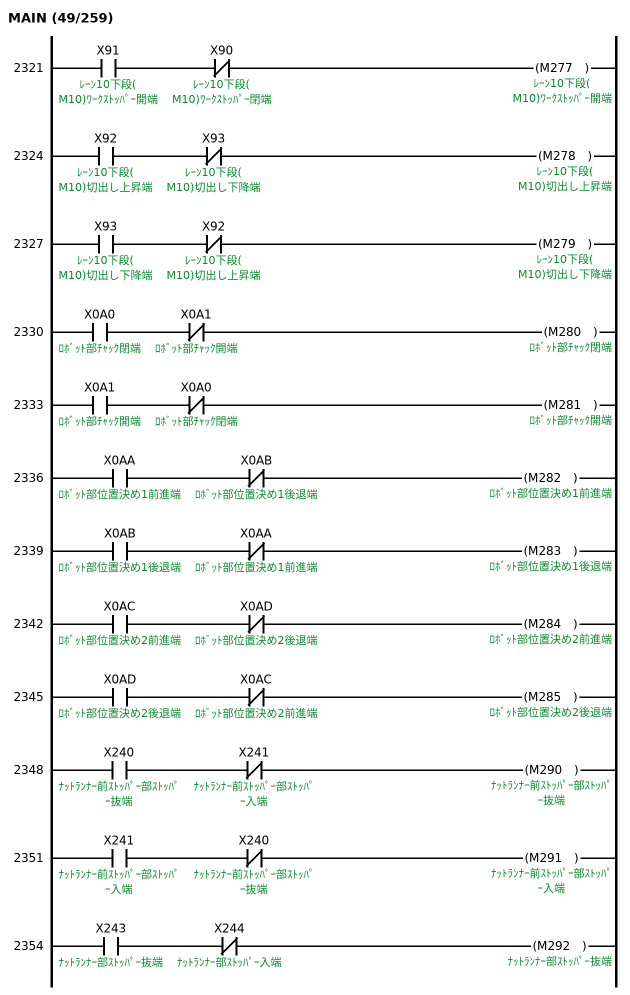
[picture p48: ladder of MAIN, rungs at steps 2321 to 2354]
2321  LD      X91  ; ﾚｰﾝ10下段(M10)ﾜｰｸｽﾄｯﾊﾟｰ開端
      ANI     X90  ; ﾚｰﾝ10下段(M10)ﾜｰｸｽﾄｯﾊﾟｰ閉端
      OUT     M277  ; ﾚｰﾝ10下段(M10)ﾜｰｸｽﾄｯﾊﾟｰ開端
2324  LD      X92  ; ﾚｰﾝ10下段(M10)切出し上昇端
      ANI     X93  ; ﾚｰﾝ10下段(M10)切出し下降端
      OUT     M278  ; ﾚｰﾝ10下段(M10)切出し上昇端
2327  LD      X93  ; ﾚｰﾝ10下段(M10)切出し下降端
      ANI     X92  ; ﾚｰﾝ10下段(M10)切出し上昇端
      OUT     M279  ; ﾚｰﾝ10下段(M10)切出し下降端
2330  LD      X0A0  ; ﾛﾎﾞｯﾄ部ﾁｬｯｸ閉端
      ANI     X0A1  ; ﾛﾎﾞｯﾄ部ﾁｬｯｸ開端
      OUT     M280  ; ﾛﾎﾞｯﾄ部ﾁｬｯｸ閉端
2333  LD      X0A1  ; ﾛﾎﾞｯﾄ部ﾁｬｯｸ開端
      ANI     X0A0  ; ﾛﾎﾞｯﾄ部ﾁｬｯｸ閉端
      OUT     M281  ; ﾛﾎﾞｯﾄ部ﾁｬｯｸ開端
2336  LD      X0AA  ; ﾛﾎﾞｯﾄ部位置決め1前進端
      ANI     X0AB  ; ﾛﾎﾞｯﾄ部位置決め1後退端
      OUT     M282  ; ﾛﾎﾞｯﾄ部位置決め1前進端
2339  LD      X0AB  ; ﾛﾎﾞｯﾄ部位置決め1後退端
      ANI     X0AA  ; ﾛﾎﾞｯﾄ部位置決め1前進端
      OUT     M283  ; ﾛﾎﾞｯﾄ部位置決め1後退端
2342  LD      X0AC  ; ﾛﾎﾞｯﾄ部位置決め2前進端
      ANI     X0AD  ; ﾛﾎﾞｯﾄ部位置決め2後退端
      OUT     M284  ; ﾛﾎﾞｯﾄ部位置決め2前進端
2345  LD      X0AD  ; ﾛﾎﾞｯﾄ部位置決め2後退端
      ANI     X0AC  ; ﾛﾎﾞｯﾄ部位置決め2前進端
      OUT     M285  ; ﾛﾎﾞｯﾄ部位置決め2後退端
2348  LD      X240  ; ﾅｯﾄﾗﾝﾅｰ前ｽﾄｯﾊﾟｰ部ｽﾄｯﾊﾟｰ抜端
      ANI     X241  ; ﾅｯﾄﾗﾝﾅｰ前ｽﾄｯﾊﾟｰ部ｽﾄｯﾊﾟｰ入端
      OUT     M290  ; ﾅｯﾄﾗﾝﾅｰ前ｽﾄｯﾊﾟｰ部ｽﾄｯﾊﾟｰ抜端
2351  LD      X241  ; ﾅｯﾄﾗﾝﾅｰ前ｽﾄｯﾊﾟｰ部ｽﾄｯﾊﾟｰ入端
      ANI     X240  ; ﾅｯﾄﾗﾝﾅｰ前ｽﾄｯﾊﾟｰ部ｽﾄｯﾊﾟｰ抜端
      OUT     M291  ; ﾅｯﾄﾗﾝﾅｰ前ｽﾄｯﾊﾟｰ部ｽﾄｯﾊﾟｰ入端
2354  LD      X243  ; ﾅｯﾄﾗﾝﾅｰ部ｽﾄｯﾊﾟｰ抜端
      ANI     X244  ; ﾅｯﾄﾗﾝﾅｰ部ｽﾄｯﾊﾟｰ入端
      OUT     M292  ; ﾅｯﾄﾗﾝﾅｰ部ｽﾄｯﾊﾟｰ抜端
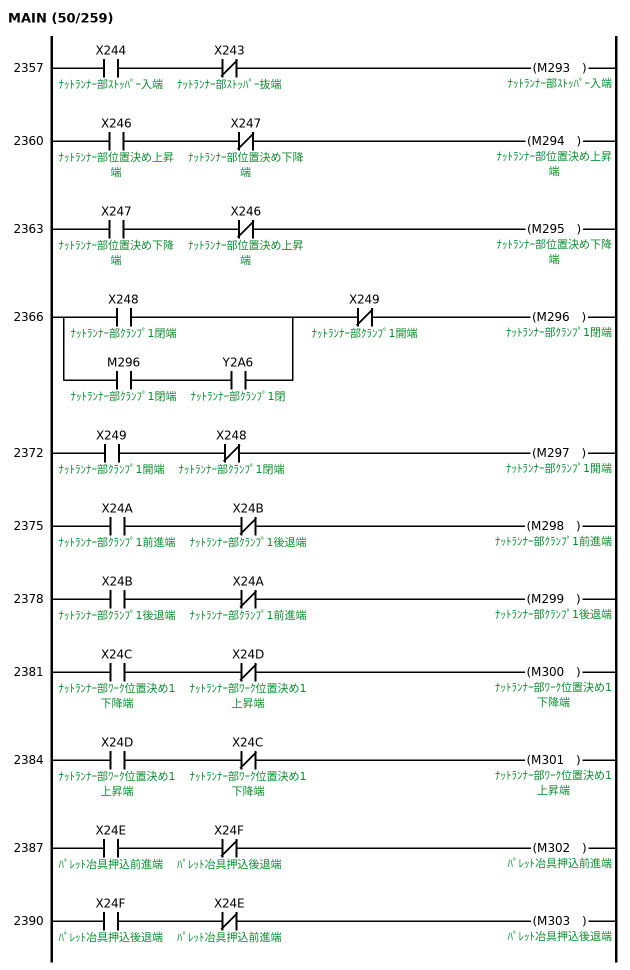
2357  LD      X244  ; ﾅｯﾄﾗﾝﾅｰ部ｽﾄｯﾊﾟｰ入端
      ANI     X243  ; ﾅｯﾄﾗﾝﾅｰ部ｽﾄｯﾊﾟｰ抜端
      OUT     M293  ; ﾅｯﾄﾗﾝﾅｰ部ｽﾄｯﾊﾟｰ入端
2360  LD      X246  ; ﾅｯﾄﾗﾝﾅｰ部位置決め上昇端
      ANI     X247  ; ﾅｯﾄﾗﾝﾅｰ部位置決め下降端
      OUT     M294  ; ﾅｯﾄﾗﾝﾅｰ部位置決め上昇端
2363  LD      X247  ; ﾅｯﾄﾗﾝﾅｰ部位置決め下降端
      ANI     X246  ; ﾅｯﾄﾗﾝﾅｰ部位置決め上昇端
      OUT     M295  ; ﾅｯﾄﾗﾝﾅｰ部位置決め下降端
2366  LD      X248  ; ﾅｯﾄﾗﾝﾅｰ部ｸﾗﾝﾌﾟ1閉端
      LD      M296  ; ﾅｯﾄﾗﾝﾅｰ部ｸﾗﾝﾌﾟ1閉端
      AND     Y2A6  ; ﾅｯﾄﾗﾝﾅｰ部ｸﾗﾝﾌﾟ1閉
      ORB
      ANI     X249  ; ﾅｯﾄﾗﾝﾅｰ部ｸﾗﾝﾌﾟ1開端
      OUT     M296  ; ﾅｯﾄﾗﾝﾅｰ部ｸﾗﾝﾌﾟ1閉端
2372  LD      X249  ; ﾅｯﾄﾗﾝﾅｰ部ｸﾗﾝﾌﾟ1開端
      ANI     X248  ; ﾅｯﾄﾗﾝﾅｰ部ｸﾗﾝﾌﾟ1閉端
      OUT     M297  ; ﾅｯﾄﾗﾝﾅｰ部ｸﾗﾝﾌﾟ1開端
2375  LD      X24A  ; ﾅｯﾄﾗﾝﾅｰ部ｸﾗﾝﾌﾟ1前進端
      ANI     X24B  ; ﾅｯﾄﾗﾝﾅｰ部ｸﾗﾝﾌﾟ1後退端
      OUT     M298  ; ﾅｯﾄﾗﾝﾅｰ部ｸﾗﾝﾌﾟ1前進端
2378  LD      X24B  ; ﾅｯﾄﾗﾝﾅｰ部ｸﾗﾝﾌﾟ1後退端
      ANI     X24A  ; ﾅｯﾄﾗﾝﾅｰ部ｸﾗﾝﾌﾟ1前進端
      OUT     M299  ; ﾅｯﾄﾗﾝﾅｰ部ｸﾗﾝﾌﾟ1後退端
2381  LD      X24C  ; ﾅｯﾄﾗﾝﾅｰ部ﾜｰｸ位置決め1下降端
      ANI     X24D  ; ﾅｯﾄﾗﾝﾅｰ部ﾜｰｸ位置決め1上昇端
      OUT     M300  ; ﾅｯﾄﾗﾝﾅｰ部ﾜｰｸ位置決め1下降端
2384  LD      X24D  ; ﾅｯﾄﾗﾝﾅｰ部ﾜｰｸ位置決め1上昇端
      ANI     X24C  ; ﾅｯﾄﾗﾝﾅｰ部ﾜｰｸ位置決め1下降端
      OUT     M301  ; ﾅｯﾄﾗﾝﾅｰ部ﾜｰｸ位置決め1上昇端
2387  LD      X24E  ; ﾊﾟﾚｯﾄ冶具押込前進端
      ANI     X24F  ; ﾊﾟﾚｯﾄ冶具押込後退端
      OUT     M302  ; ﾊﾟﾚｯﾄ冶具押込前進端
2390  LD      X24F  ; ﾊﾟﾚｯﾄ冶具押込後退端
      ANI     X24E  ; ﾊﾟﾚｯﾄ冶具押込前進端
      OUT     M303  ; ﾊﾟﾚｯﾄ冶具押込後退端
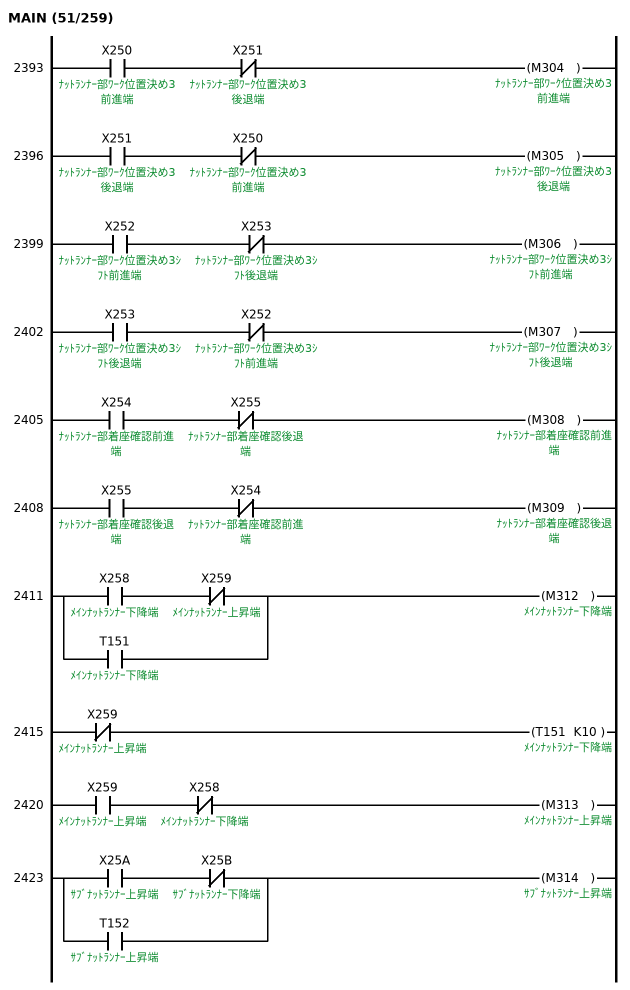
2393  LD      X250  ; ﾅｯﾄﾗﾝﾅｰ部ﾜｰｸ位置決め3前進端
      ANI     X251  ; ﾅｯﾄﾗﾝﾅｰ部ﾜｰｸ位置決め3後退端
      OUT     M304  ; ﾅｯﾄﾗﾝﾅｰ部ﾜｰｸ位置決め3前進端
2396  LD      X251  ; ﾅｯﾄﾗﾝﾅｰ部ﾜｰｸ位置決め3後退端
      ANI     X250  ; ﾅｯﾄﾗﾝﾅｰ部ﾜｰｸ位置決め3前進端
      OUT     M305  ; ﾅｯﾄﾗﾝﾅｰ部ﾜｰｸ位置決め3後退端
2399  LD      X252  ; ﾅｯﾄﾗﾝﾅｰ部ﾜｰｸ位置決め3ｼﾌﾄ前進端
      ANI     X253  ; ﾅｯﾄﾗﾝﾅｰ部ﾜｰｸ位置決め3ｼﾌﾄ後退端
      OUT     M306  ; ﾅｯﾄﾗﾝﾅｰ部ﾜｰｸ位置決め3ｼﾌﾄ前進端
2402  LD      X253  ; ﾅｯﾄﾗﾝﾅｰ部ﾜｰｸ位置決め3ｼﾌﾄ後退端
      ANI     X252  ; ﾅｯﾄﾗﾝﾅｰ部ﾜｰｸ位置決め3ｼﾌﾄ前進端
      OUT     M307  ; ﾅｯﾄﾗﾝﾅｰ部ﾜｰｸ位置決め3ｼﾌﾄ後退端
2405  LD      X254  ; ﾅｯﾄﾗﾝﾅｰ部着座確認前進端
      ANI     X255  ; ﾅｯﾄﾗﾝﾅｰ部着座確認後退端
      OUT     M308  ; ﾅｯﾄﾗﾝﾅｰ部着座確認前進端
2408  LD      X255  ; ﾅｯﾄﾗﾝﾅｰ部着座確認後退端
      ANI     X254  ; ﾅｯﾄﾗﾝﾅｰ部着座確認前進端
      OUT     M309  ; ﾅｯﾄﾗﾝﾅｰ部着座確認後退端
2411  LD      X258  ; ﾒｲﾝﾅｯﾄﾗﾝﾅｰ下降端
      ANI     X259  ; ﾒｲﾝﾅｯﾄﾗﾝﾅｰ上昇端
      OR      T151  ; ﾒｲﾝﾅｯﾄﾗﾝﾅｰ下降端
      OUT     M312  ; ﾒｲﾝﾅｯﾄﾗﾝﾅｰ下降端
2415  LDI     X259  ; ﾒｲﾝﾅｯﾄﾗﾝﾅｰ上昇端
      OUT     T151 K10  ; ﾒｲﾝﾅｯﾄﾗﾝﾅｰ下降端
2420  LD      X259  ; ﾒｲﾝﾅｯﾄﾗﾝﾅｰ上昇端
      ANI     X258  ; ﾒｲﾝﾅｯﾄﾗﾝﾅｰ下降端
      OUT     M313  ; ﾒｲﾝﾅｯﾄﾗﾝﾅｰ上昇端
2423  LD      X25A  ; ｻﾌﾞﾅｯﾄﾗﾝﾅｰ上昇端
      ANI     X25B  ; ｻﾌﾞﾅｯﾄﾗﾝﾅｰ下降端
      OR      T152  ; ｻﾌﾞﾅｯﾄﾗﾝﾅｰ上昇端
      OUT     M314  ; ｻﾌﾞﾅｯﾄﾗﾝﾅｰ上昇端
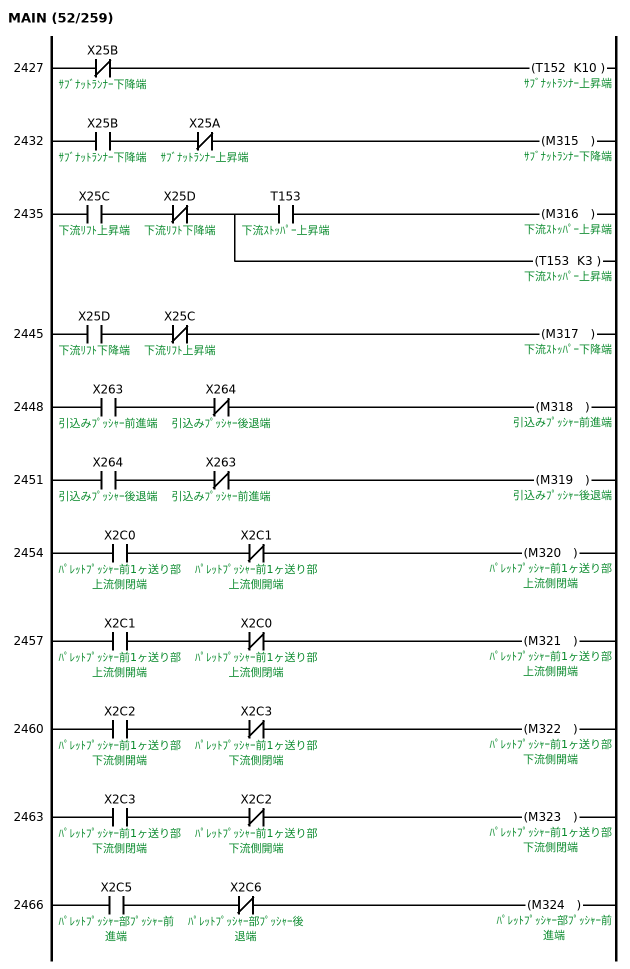
2427  LDI     X25B  ; ｻﾌﾞﾅｯﾄﾗﾝﾅｰ下降端
      OUT     T152 K10  ; ｻﾌﾞﾅｯﾄﾗﾝﾅｰ上昇端
2432  LD      X25B  ; ｻﾌﾞﾅｯﾄﾗﾝﾅｰ下降端
      ANI     X25A  ; ｻﾌﾞﾅｯﾄﾗﾝﾅｰ上昇端
      OUT     M315  ; ｻﾌﾞﾅｯﾄﾗﾝﾅｰ下降端
2435  LD      X25C  ; 下流ﾘﾌﾄ上昇端
      ANI     X25D  ; 下流ﾘﾌﾄ下降端
      MPS
      AND     T153  ; 下流ｽﾄｯﾊﾟｰ上昇端
      OUT     M316  ; 下流ｽﾄｯﾊﾟｰ上昇端
      MPP
      OUT     T153 K3  ; 下流ｽﾄｯﾊﾟｰ上昇端
2445  LD      X25D  ; 下流ﾘﾌﾄ下降端
      ANI     X25C  ; 下流ﾘﾌﾄ上昇端
      OUT     M317  ; 下流ｽﾄｯﾊﾟｰ下降端
2448  LD      X263  ; 引込みﾌﾟｯｼｬｰ前進端
      ANI     X264  ; 引込みﾌﾟｯｼｬｰ後退端
      OUT     M318  ; 引込みﾌﾟｯｼｬｰ前進端
2451  LD      X264  ; 引込みﾌﾟｯｼｬｰ後退端
      ANI     X263  ; 引込みﾌﾟｯｼｬｰ前進端
      OUT     M319  ; 引込みﾌﾟｯｼｬｰ後退端
2454  LD      X2C0  ; ﾊﾟﾚｯﾄﾌﾟｯｼｬｰ前1ヶ送り部上流側閉端
      ANI     X2C1  ; ﾊﾟﾚｯﾄﾌﾟｯｼｬｰ前1ヶ送り部上流側開端
      OUT     M320  ; ﾊﾟﾚｯﾄﾌﾟｯｼｬｰ前1ヶ送り部上流側閉端
2457  LD      X2C1  ; ﾊﾟﾚｯﾄﾌﾟｯｼｬｰ前1ヶ送り部上流側開端
      ANI     X2C0  ; ﾊﾟﾚｯﾄﾌﾟｯｼｬｰ前1ヶ送り部上流側閉端
      OUT     M321  ; ﾊﾟﾚｯﾄﾌﾟｯｼｬｰ前1ヶ送り部上流側開端
2460  LD      X2C2  ; ﾊﾟﾚｯﾄﾌﾟｯｼｬｰ前1ヶ送り部下流側開端
      ANI     X2C3  ; ﾊﾟﾚｯﾄﾌﾟｯｼｬｰ前1ヶ送り部下流側閉端
      OUT     M322  ; ﾊﾟﾚｯﾄﾌﾟｯｼｬｰ前1ヶ送り部下流側開端
2463  LD      X2C3  ; ﾊﾟﾚｯﾄﾌﾟｯｼｬｰ前1ヶ送り部下流側閉端
      ANI     X2C2  ; ﾊﾟﾚｯﾄﾌﾟｯｼｬｰ前1ヶ送り部下流側開端
      OUT     M323  ; ﾊﾟﾚｯﾄﾌﾟｯｼｬｰ前1ヶ送り部下流側閉端
2466  LD      X2C5  ; ﾊﾟﾚｯﾄﾌﾟｯｼｬｰ部ﾌﾟｯｼｬｰ前進端
      ANI     X2C6  ; ﾊﾟﾚｯﾄﾌﾟｯｼｬｰ部ﾌﾟｯｼｬｰ後退端
      OUT     M324  ; ﾊﾟﾚｯﾄﾌﾟｯｼｬｰ部ﾌﾟｯｼｬｰ前進端
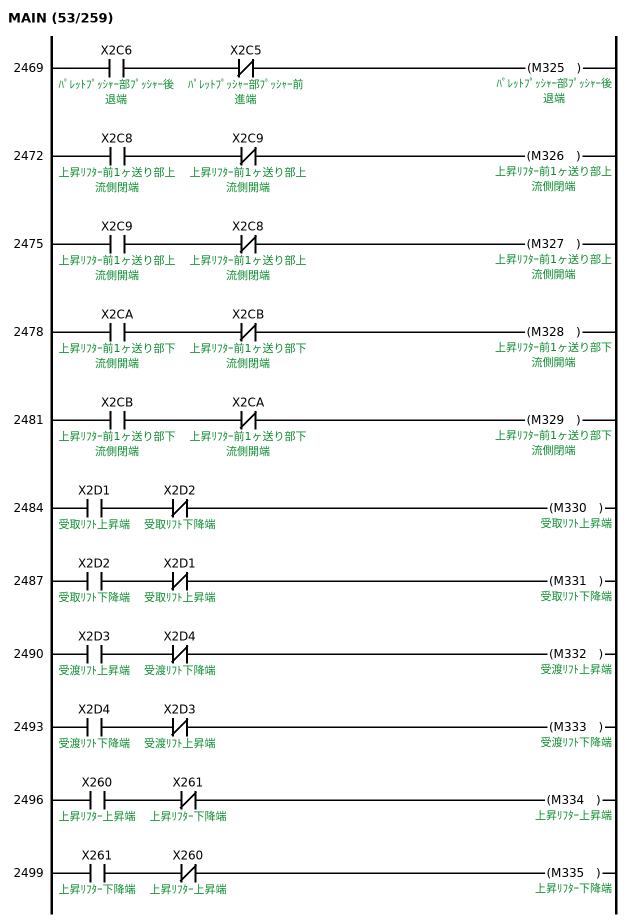
2469  LD      X2C6  ; ﾊﾟﾚｯﾄﾌﾟｯｼｬｰ部ﾌﾟｯｼｬｰ後退端
      ANI     X2C5  ; ﾊﾟﾚｯﾄﾌﾟｯｼｬｰ部ﾌﾟｯｼｬｰ前進端
      OUT     M325  ; ﾊﾟﾚｯﾄﾌﾟｯｼｬｰ部ﾌﾟｯｼｬｰ後退端
2472  LD      X2C8  ; 上昇ﾘﾌﾀｰ前1ヶ送り部上流側閉端
      ANI     X2C9  ; 上昇ﾘﾌﾀｰ前1ヶ送り部上流側開端
      OUT     M326  ; 上昇ﾘﾌﾀｰ前1ヶ送り部上流側閉端
2475  LD      X2C9  ; 上昇ﾘﾌﾀｰ前1ヶ送り部上流側開端
      ANI     X2C8  ; 上昇ﾘﾌﾀｰ前1ヶ送り部上流側閉端
      OUT     M327  ; 上昇ﾘﾌﾀｰ前1ヶ送り部上流側開端
2478  LD      X2CA  ; 上昇ﾘﾌﾀｰ前1ヶ送り部下流側開端
      ANI     X2CB  ; 上昇ﾘﾌﾀｰ前1ヶ送り部下流側閉端
      OUT     M328  ; 上昇ﾘﾌﾀｰ前1ヶ送り部下流側開端
2481  LD      X2CB  ; 上昇ﾘﾌﾀｰ前1ヶ送り部下流側閉端
      ANI     X2CA  ; 上昇ﾘﾌﾀｰ前1ヶ送り部下流側開端
      OUT     M329  ; 上昇ﾘﾌﾀｰ前1ヶ送り部下流側閉端
2484  LD      X2D1  ; 受取ﾘﾌﾄ上昇端
      ANI     X2D2  ; 受取ﾘﾌﾄ下降端
      OUT     M330  ; 受取ﾘﾌﾄ上昇端
2487  LD      X2D2  ; 受取ﾘﾌﾄ下降端
      ANI     X2D1  ; 受取ﾘﾌﾄ上昇端
      OUT     M331  ; 受取ﾘﾌﾄ下降端
2490  LD      X2D3  ; 受渡ﾘﾌﾄ上昇端
      ANI     X2D4  ; 受渡ﾘﾌﾄ下降端
      OUT     M332  ; 受渡ﾘﾌﾄ上昇端
2493  LD      X2D4  ; 受渡ﾘﾌﾄ下降端
      ANI     X2D3  ; 受渡ﾘﾌﾄ上昇端
      OUT     M333  ; 受渡ﾘﾌﾄ下降端
2496  LD      X260  ; 上昇ﾘﾌﾀｰ上昇端
      ANI     X261  ; 上昇ﾘﾌﾀｰ下降端
      OUT     M334  ; 上昇ﾘﾌﾀｰ上昇端
2499  LD      X261  ; 上昇ﾘﾌﾀｰ下降端
      ANI     X260  ; 上昇ﾘﾌﾀｰ上昇端
      OUT     M335  ; 上昇ﾘﾌﾀｰ下降端
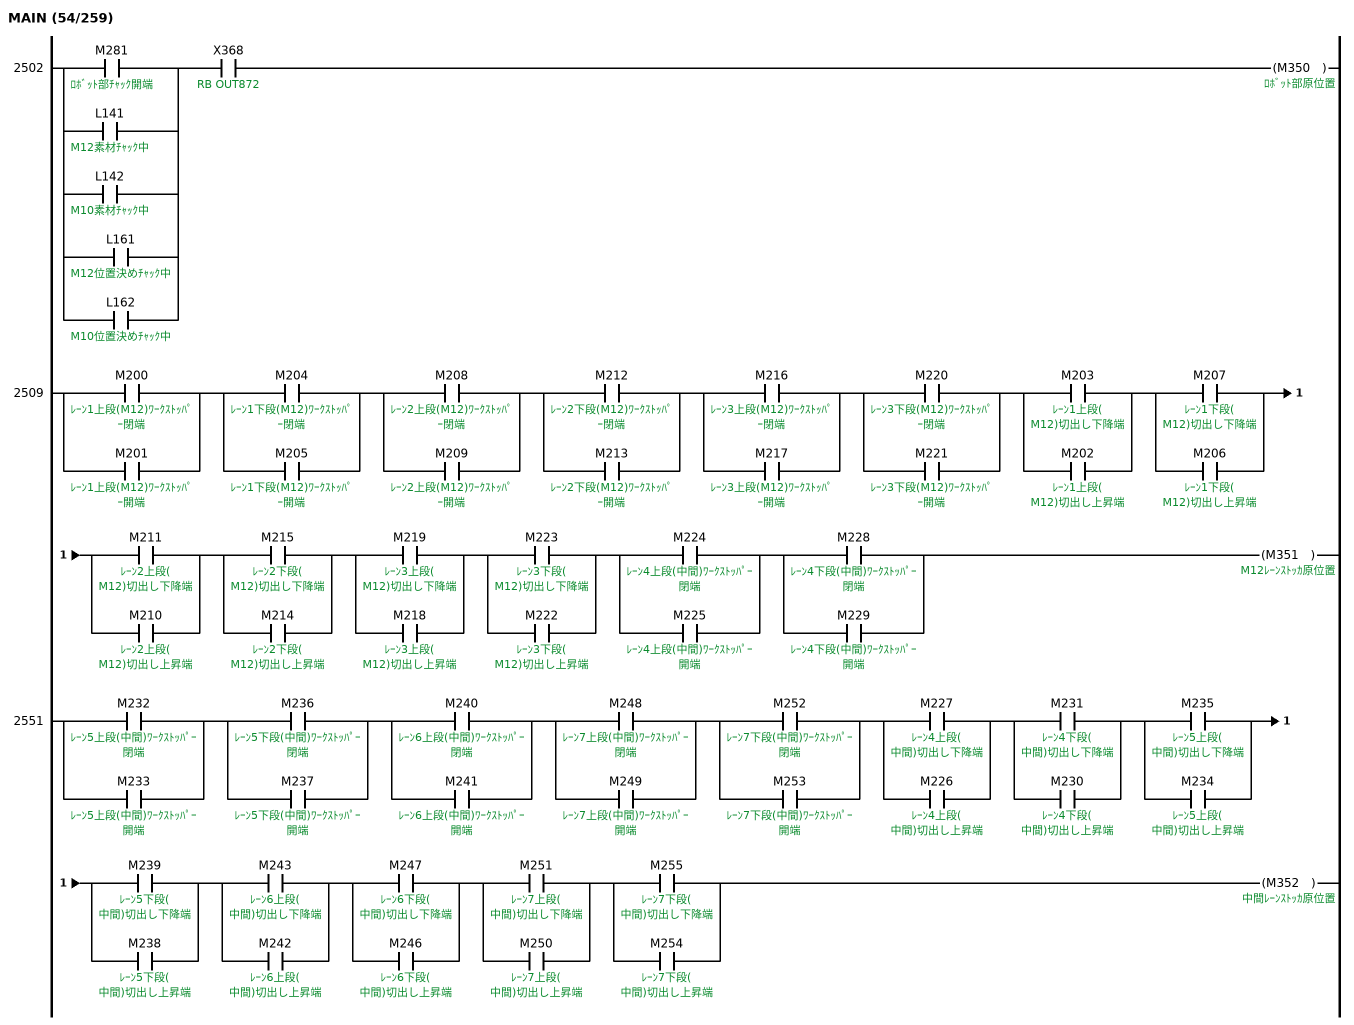
2502  LD      M281  ; ﾛﾎﾞｯﾄ部ﾁｬｯｸ開端
      OR      L141  ; M12素材ﾁｬｯｸ中
      OR      L142  ; M10素材ﾁｬｯｸ中
      OR      L161  ; M12位置決めﾁｬｯｸ中
      OR      L162  ; M10位置決めﾁｬｯｸ中
      AND     X368  ; RB OUT872
      OUT     M350  ; ﾛﾎﾞｯﾄ部原位置
2509  LD      M200  ; ﾚｰﾝ1上段(M12)ﾜｰｸｽﾄｯﾊﾟｰ閉端
      OR      M201  ; ﾚｰﾝ1上段(M12)ﾜｰｸｽﾄｯﾊﾟｰ開端
      LD      M204  ; ﾚｰﾝ1下段(M12)ﾜｰｸｽﾄｯﾊﾟｰ閉端
      OR      M205  ; ﾚｰﾝ1下段(M12)ﾜｰｸｽﾄｯﾊﾟｰ開端
      ANB
      LD      M208  ; ﾚｰﾝ2上段(M12)ﾜｰｸｽﾄｯﾊﾟｰ閉端
      OR      M209  ; ﾚｰﾝ2上段(M12)ﾜｰｸｽﾄｯﾊﾟｰ開端
      ANB
      LD      M212  ; ﾚｰﾝ2下段(M12)ﾜｰｸｽﾄｯﾊﾟｰ閉端
      OR      M213  ; ﾚｰﾝ2下段(M12)ﾜｰｸｽﾄｯﾊﾟｰ開端
      ANB
      LD      M216  ; ﾚｰﾝ3上段(M12)ﾜｰｸｽﾄｯﾊﾟｰ閉端
      OR      M217  ; ﾚｰﾝ3上段(M12)ﾜｰｸｽﾄｯﾊﾟｰ開端
      ANB
      LD      M220  ; ﾚｰﾝ3下段(M12)ﾜｰｸｽﾄｯﾊﾟｰ閉端
      OR      M221  ; ﾚｰﾝ3下段(M12)ﾜｰｸｽﾄｯﾊﾟｰ開端
      ANB
      LD      M203  ; ﾚｰﾝ1上段(M12)切出し下降端
      OR      M202  ; ﾚｰﾝ1上段(M12)切出し上昇端
      ANB
      LD      M207  ; ﾚｰﾝ1下段(M12)切出し下降端
      OR      M206  ; ﾚｰﾝ1下段(M12)切出し上昇端
      ANB
      LD      M211  ; ﾚｰﾝ2上段(M12)切出し下降端
      OR      M210  ; ﾚｰﾝ2上段(M12)切出し上昇端
      ANB
      LD      M215  ; ﾚｰﾝ2下段(M12)切出し下降端
      OR      M214  ; ﾚｰﾝ2下段(M12)切出し上昇端
      ANB
      LD      M219  ; ﾚｰﾝ3上段(M12)切出し下降端
      OR      M218  ; ﾚｰﾝ3上段(M12)切出し上昇端
      ANB
      LD      M223  ; ﾚｰﾝ3下段(M12)切出し下降端
      OR      M222  ; ﾚｰﾝ3下段(M12)切出し上昇端
      ANB
      LD      M224  ; ﾚｰﾝ4上段(中間)ﾜｰｸｽﾄｯﾊﾟｰ閉端
      OR      M225  ; ﾚｰﾝ4上段(中間)ﾜｰｸｽﾄｯﾊﾟｰ開端
      ANB
      LD      M228  ; ﾚｰﾝ4下段(中間)ﾜｰｸｽﾄｯﾊﾟｰ閉端
      OR      M229  ; ﾚｰﾝ4下段(中間)ﾜｰｸｽﾄｯﾊﾟｰ開端
      ANB
      OUT     M351  ; M12ﾚｰﾝｽﾄｯｶ原位置
2551  LD      M232  ; ﾚｰﾝ5上段(中間)ﾜｰｸｽﾄｯﾊﾟｰ閉端
      OR      M233  ; ﾚｰﾝ5上段(中間)ﾜｰｸｽﾄｯﾊﾟｰ開端
      LD      M236  ; ﾚｰﾝ5下段(中間)ﾜｰｸｽﾄｯﾊﾟｰ閉端
      OR      M237  ; ﾚｰﾝ5下段(中間)ﾜｰｸｽﾄｯﾊﾟｰ開端
      ANB
      LD      M240  ; ﾚｰﾝ6上段(中間)ﾜｰｸｽﾄｯﾊﾟｰ閉端
      OR      M241  ; ﾚｰﾝ6上段(中間)ﾜｰｸｽﾄｯﾊﾟｰ開端
      ANB
      LD      M248  ; ﾚｰﾝ7上段(中間)ﾜｰｸｽﾄｯﾊﾟｰ閉端
      OR      M249  ; ﾚｰﾝ7上段(中間)ﾜｰｸｽﾄｯﾊﾟｰ開端
      ANB
      LD      M252  ; ﾚｰﾝ7下段(中間)ﾜｰｸｽﾄｯﾊﾟｰ閉端
      OR      M253  ; ﾚｰﾝ7下段(中間)ﾜｰｸｽﾄｯﾊﾟｰ開端
      ANB
      LD      M227  ; ﾚｰﾝ4上段(中間)切出し下降端
      OR      M226  ; ﾚｰﾝ4上段(中間)切出し上昇端
      ANB
      LD      M231  ; ﾚｰﾝ4下段(中間)切出し下降端
      OR      M230  ; ﾚｰﾝ4下段(中間)切出し上昇端
      ANB
      LD      M235  ; ﾚｰﾝ5上段(中間)切出し下降端
      OR      M234  ; ﾚｰﾝ5上段(中間)切出し上昇端
      ANB
      LD      M239  ; ﾚｰﾝ5下段(中間)切出し下降端
      OR      M238  ; ﾚｰﾝ5下段(中間)切出し上昇端
      ANB
      LD      M243  ; ﾚｰﾝ6上段(中間)切出し下降端
      OR      M242  ; ﾚｰﾝ6上段(中間)切出し上昇端
      ANB
      LD      M247  ; ﾚｰﾝ6下段(中間)切出し下降端
      OR      M246  ; ﾚｰﾝ6下段(中間)切出し上昇端
      ANB
      LD      M251  ; ﾚｰﾝ7上段(中間)切出し下降端
      OR      M250  ; ﾚｰﾝ7上段(中間)切出し上昇端
      ANB
      LD      M255  ; ﾚｰﾝ7下段(中間)切出し下降端
      OR      M254  ; ﾚｰﾝ7下段(中間)切出し上昇端
      ANB
      OUT     M352  ; 中間ﾚｰﾝｽﾄｯｶ原位置
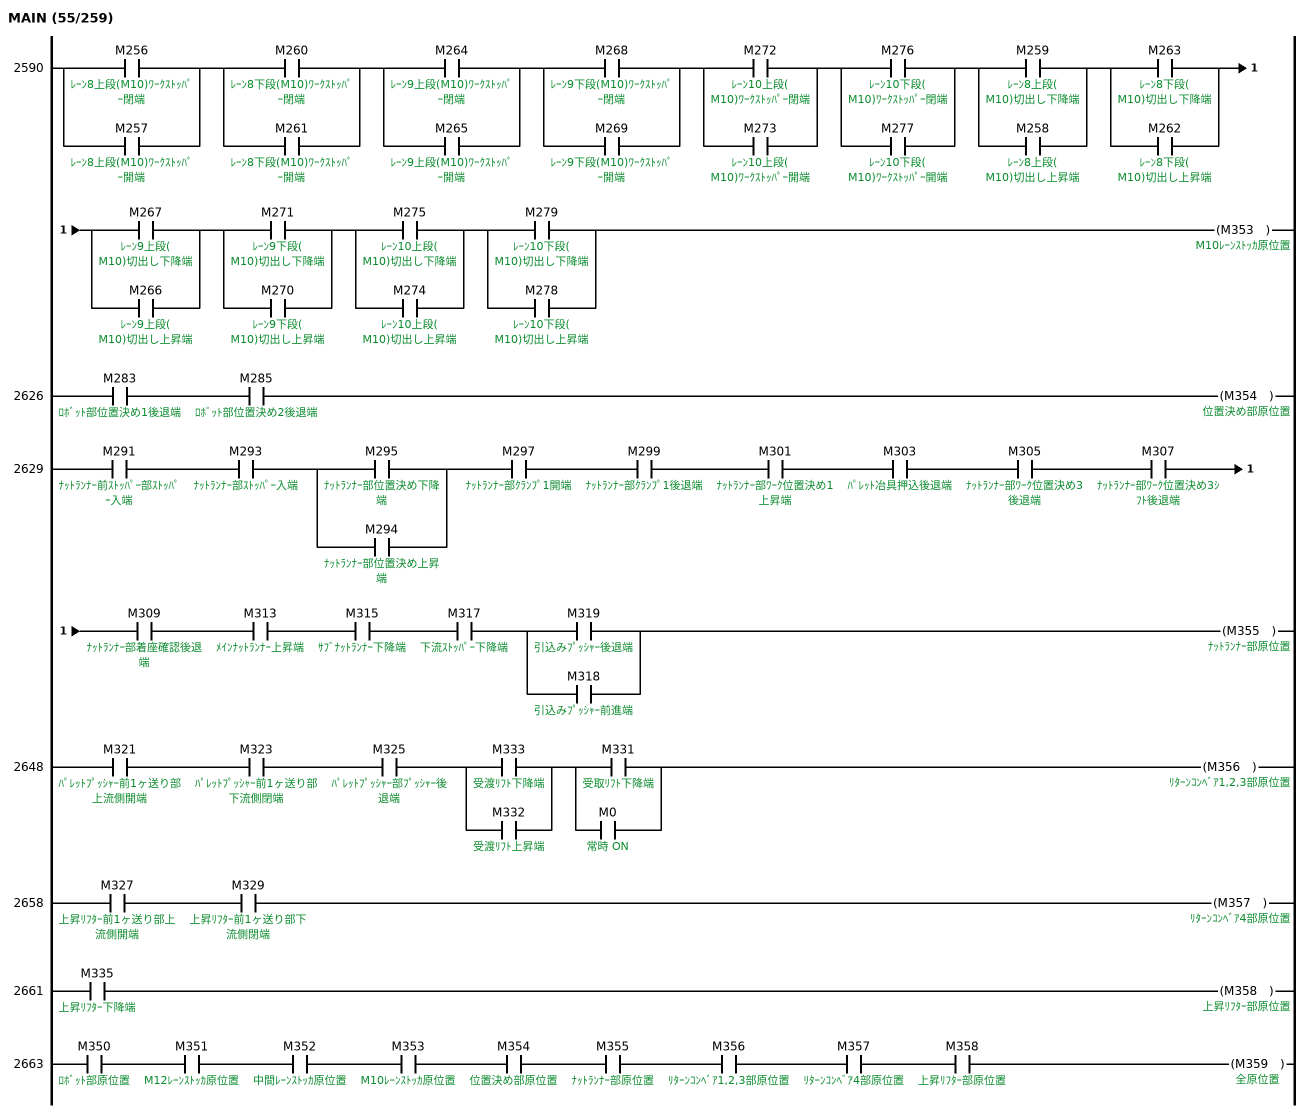
2590  LD      M256  ; ﾚｰﾝ8上段(M10)ﾜｰｸｽﾄｯﾊﾟｰ閉端
      OR      M257  ; ﾚｰﾝ8上段(M10)ﾜｰｸｽﾄｯﾊﾟｰ開端
      LD      M260  ; ﾚｰﾝ8下段(M10)ﾜｰｸｽﾄｯﾊﾟｰ閉端
      OR      M261  ; ﾚｰﾝ8下段(M10)ﾜｰｸｽﾄｯﾊﾟｰ開端
      ANB
      LD      M264  ; ﾚｰﾝ9上段(M10)ﾜｰｸｽﾄｯﾊﾟｰ閉端
      OR      M265  ; ﾚｰﾝ9上段(M10)ﾜｰｸｽﾄｯﾊﾟｰ開端
      ANB
      LD      M268  ; ﾚｰﾝ9下段(M10)ﾜｰｸｽﾄｯﾊﾟｰ閉端
      OR      M269  ; ﾚｰﾝ9下段(M10)ﾜｰｸｽﾄｯﾊﾟｰ開端
      ANB
      LD      M272  ; ﾚｰﾝ10上段(M10)ﾜｰｸｽﾄｯﾊﾟｰ閉端
      OR      M273  ; ﾚｰﾝ10上段(M10)ﾜｰｸｽﾄｯﾊﾟｰ開端
      ANB
      LD      M276  ; ﾚｰﾝ10下段(M10)ﾜｰｸｽﾄｯﾊﾟｰ閉端
      OR      M277  ; ﾚｰﾝ10下段(M10)ﾜｰｸｽﾄｯﾊﾟｰ開端
      ANB
      LD      M259  ; ﾚｰﾝ8上段(M10)切出し下降端
      OR      M258  ; ﾚｰﾝ8上段(M10)切出し上昇端
      ANB
      LD      M263  ; ﾚｰﾝ8下段(M10)切出し下降端
      OR      M262  ; ﾚｰﾝ8下段(M10)切出し上昇端
      ANB
      LD      M267  ; ﾚｰﾝ9上段(M10)切出し下降端
      OR      M266  ; ﾚｰﾝ9上段(M10)切出し上昇端
      ANB
      LD      M271  ; ﾚｰﾝ9下段(M10)切出し下降端
      OR      M270  ; ﾚｰﾝ9下段(M10)切出し上昇端
      ANB
      LD      M275  ; ﾚｰﾝ10上段(M10)切出し下降端
      OR      M274  ; ﾚｰﾝ10上段(M10)切出し上昇端
      ANB
      LD      M279  ; ﾚｰﾝ10下段(M10)切出し下降端
      OR      M278  ; ﾚｰﾝ10下段(M10)切出し上昇端
      ANB
      OUT     M353  ; M10ﾚｰﾝｽﾄｯｶ原位置
2626  LD      M283  ; ﾛﾎﾞｯﾄ部位置決め1後退端
      AND     M285  ; ﾛﾎﾞｯﾄ部位置決め2後退端
      OUT     M354  ; 位置決め部原位置
2629  LD      M291  ; ﾅｯﾄﾗﾝﾅｰ前ｽﾄｯﾊﾟｰ部ｽﾄｯﾊﾟｰ入端
      AND     M293  ; ﾅｯﾄﾗﾝﾅｰ部ｽﾄｯﾊﾟｰ入端
      LD      M295  ; ﾅｯﾄﾗﾝﾅｰ部位置決め下降端
      OR      M294  ; ﾅｯﾄﾗﾝﾅｰ部位置決め上昇端
      ANB
      AND     M297  ; ﾅｯﾄﾗﾝﾅｰ部ｸﾗﾝﾌﾟ1開端
      AND     M299  ; ﾅｯﾄﾗﾝﾅｰ部ｸﾗﾝﾌﾟ1後退端
      AND     M301  ; ﾅｯﾄﾗﾝﾅｰ部ﾜｰｸ位置決め1上昇端
      AND     M303  ; ﾊﾟﾚｯﾄ冶具押込後退端
      AND     M305  ; ﾅｯﾄﾗﾝﾅｰ部ﾜｰｸ位置決め3後退端
      AND     M307  ; ﾅｯﾄﾗﾝﾅｰ部ﾜｰｸ位置決め3ｼﾌﾄ後退端
      AND     M309  ; ﾅｯﾄﾗﾝﾅｰ部着座確認後退端
      AND     M313  ; ﾒｲﾝﾅｯﾄﾗﾝﾅｰ上昇端
      AND     M315  ; ｻﾌﾞﾅｯﾄﾗﾝﾅｰ下降端
      AND     M317  ; 下流ｽﾄｯﾊﾟｰ下降端
      LD      M319  ; 引込みﾌﾟｯｼｬｰ後退端
      OR      M318  ; 引込みﾌﾟｯｼｬｰ前進端
      ANB
      OUT     M355  ; ﾅｯﾄﾗﾝﾅｰ部原位置
2648  LD      M321  ; ﾊﾟﾚｯﾄﾌﾟｯｼｬｰ前1ヶ送り部上流側開端
      AND     M323  ; ﾊﾟﾚｯﾄﾌﾟｯｼｬｰ前1ヶ送り部下流側閉端
      AND     M325  ; ﾊﾟﾚｯﾄﾌﾟｯｼｬｰ部ﾌﾟｯｼｬｰ後退端
      LD      M333  ; 受渡ﾘﾌﾄ下降端
      OR      M332  ; 受渡ﾘﾌﾄ上昇端
      ANB
      LD      M331  ; 受取ﾘﾌﾄ下降端
      OR      M0  ; 常時 ON
      ANB
      OUT     M356  ; ﾘﾀｰﾝｺﾝﾍﾞｱ1,2,3部原位置
2658  LD      M327  ; 上昇ﾘﾌﾀｰ前1ヶ送り部上流側開端
      AND     M329  ; 上昇ﾘﾌﾀｰ前1ヶ送り部下流側閉端
      OUT     M357  ; ﾘﾀｰﾝｺﾝﾍﾞｱ4部原位置
2661  LD      M335  ; 上昇ﾘﾌﾀｰ下降端
      OUT     M358  ; 上昇ﾘﾌﾀｰ部原位置
2663  LD      M350  ; ﾛﾎﾞｯﾄ部原位置
      AND     M351  ; M12ﾚｰﾝｽﾄｯｶ原位置
      AND     M352  ; 中間ﾚｰﾝｽﾄｯｶ原位置
      AND     M353  ; M10ﾚｰﾝｽﾄｯｶ原位置
      AND     M354  ; 位置決め部原位置
      AND     M355  ; ﾅｯﾄﾗﾝﾅｰ部原位置
      AND     M356  ; ﾘﾀｰﾝｺﾝﾍﾞｱ1,2,3部原位置
      AND     M357  ; ﾘﾀｰﾝｺﾝﾍﾞｱ4部原位置
      AND     M358  ; 上昇ﾘﾌﾀｰ部原位置
      OUT     M359  ; 全原位置
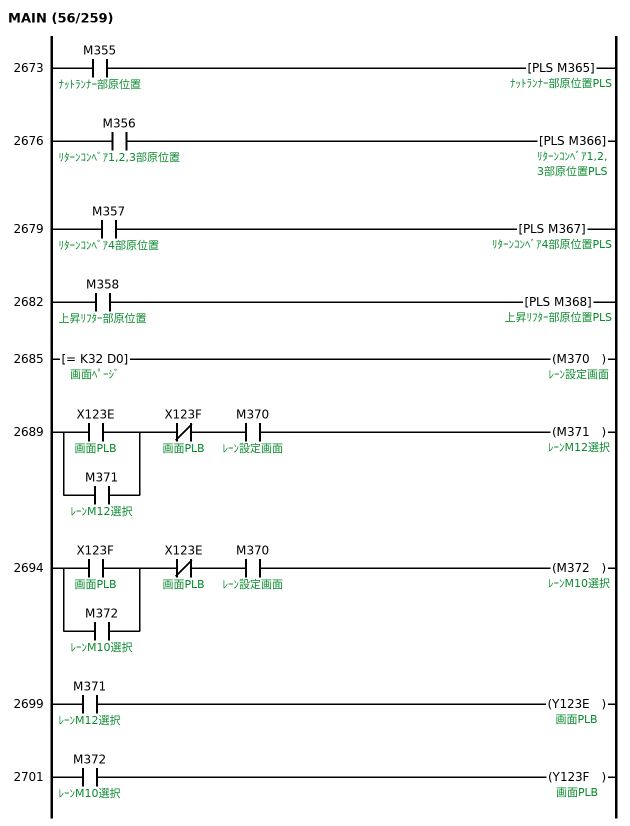
2673  LD      M355  ; ﾅｯﾄﾗﾝﾅｰ部原位置
      PLS     M365  ; ﾅｯﾄﾗﾝﾅｰ部原位置PLS
2676  LD      M356  ; ﾘﾀｰﾝｺﾝﾍﾞｱ1,2,3部原位置
      PLS     M366  ; ﾘﾀｰﾝｺﾝﾍﾞｱ1,2,3部原位置PLS
2679  LD      M357  ; ﾘﾀｰﾝｺﾝﾍﾞｱ4部原位置
      PLS     M367  ; ﾘﾀｰﾝｺﾝﾍﾞｱ4部原位置PLS
2682  LD      M358  ; 上昇ﾘﾌﾀｰ部原位置
      PLS     M368  ; 上昇ﾘﾌﾀｰ部原位置PLS
2685  LD=     K32 D0  ; 画面ﾍﾟｰｼﾞ
      OUT     M370  ; ﾚｰﾝ設定画面
2689  LD      X123E  ; 画面PLB
      OR      M371  ; ﾚｰﾝM12選択
      ANI     X123F  ; 画面PLB
      AND     M370  ; ﾚｰﾝ設定画面
      OUT     M371  ; ﾚｰﾝM12選択
2694  LD      X123F  ; 画面PLB
      OR      M372  ; ﾚｰﾝM10選択
      ANI     X123E  ; 画面PLB
      AND     M370  ; ﾚｰﾝ設定画面
      OUT     M372  ; ﾚｰﾝM10選択
2699  LD      M371  ; ﾚｰﾝM12選択
      OUT     Y123E  ; 画面PLB
2701  LD      M372  ; ﾚｰﾝM10選択
      OUT     Y123F  ; 画面PLB
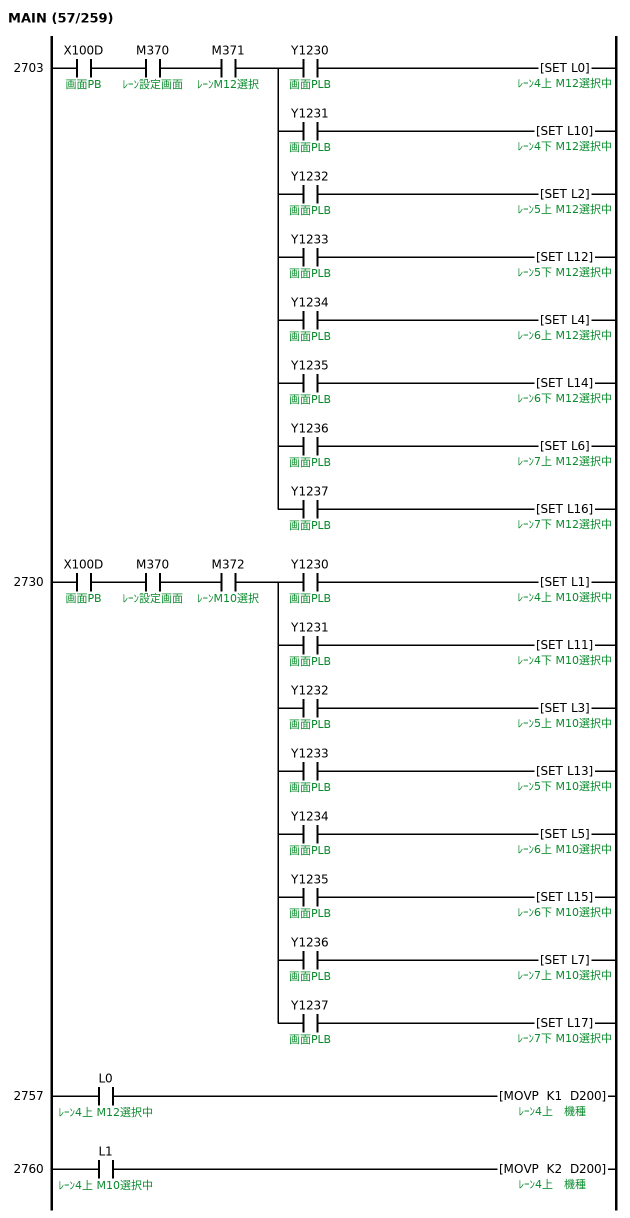
2703  LD      X100D  ; 画面PB
      AND     M370  ; ﾚｰﾝ設定画面
      AND     M371  ; ﾚｰﾝM12選択
      MPS
      AND     Y1230  ; 画面PLB
      SET     L0  ; ﾚｰﾝ4上 M12選択中
      MRD
      AND     Y1231  ; 画面PLB
      SET     L10  ; ﾚｰﾝ4下 M12選択中
      MRD
      AND     Y1232  ; 画面PLB
      SET     L2  ; ﾚｰﾝ5上 M12選択中
      MRD
      AND     Y1233  ; 画面PLB
      SET     L12  ; ﾚｰﾝ5下 M12選択中
      MRD
      AND     Y1234  ; 画面PLB
      SET     L4  ; ﾚｰﾝ6上 M12選択中
      MRD
      AND     Y1235  ; 画面PLB
      SET     L14  ; ﾚｰﾝ6下 M12選択中
      MRD
      AND     Y1236  ; 画面PLB
      SET     L6  ; ﾚｰﾝ7上 M12選択中
      MPP
      AND     Y1237  ; 画面PLB
      SET     L16  ; ﾚｰﾝ7下 M12選択中
2730  LD      X100D  ; 画面PB
      AND     M370  ; ﾚｰﾝ設定画面
      AND     M372  ; ﾚｰﾝM10選択
      MPS
      AND     Y1230  ; 画面PLB
      SET     L1  ; ﾚｰﾝ4上 M10選択中
      MRD
      AND     Y1231  ; 画面PLB
      SET     L11  ; ﾚｰﾝ4下 M10選択中
      MRD
      AND     Y1232  ; 画面PLB
      SET     L3  ; ﾚｰﾝ5上 M10選択中
      MRD
      AND     Y1233  ; 画面PLB
      SET     L13  ; ﾚｰﾝ5下 M10選択中
      MRD
      AND     Y1234  ; 画面PLB
      SET     L5  ; ﾚｰﾝ6上 M10選択中
      MRD
      AND     Y1235  ; 画面PLB
      SET     L15  ; ﾚｰﾝ6下 M10選択中
      MRD
      AND     Y1236  ; 画面PLB
      SET     L7  ; ﾚｰﾝ7上 M10選択中
      MPP
      AND     Y1237  ; 画面PLB
      SET     L17  ; ﾚｰﾝ7下 M10選択中
2757  LD      L0  ; ﾚｰﾝ4上 M12選択中
      MOVP    K1 D200  ; ﾚｰﾝ4上　機種
2760  LD      L1  ; ﾚｰﾝ4上 M10選択中
      MOVP    K2 D200
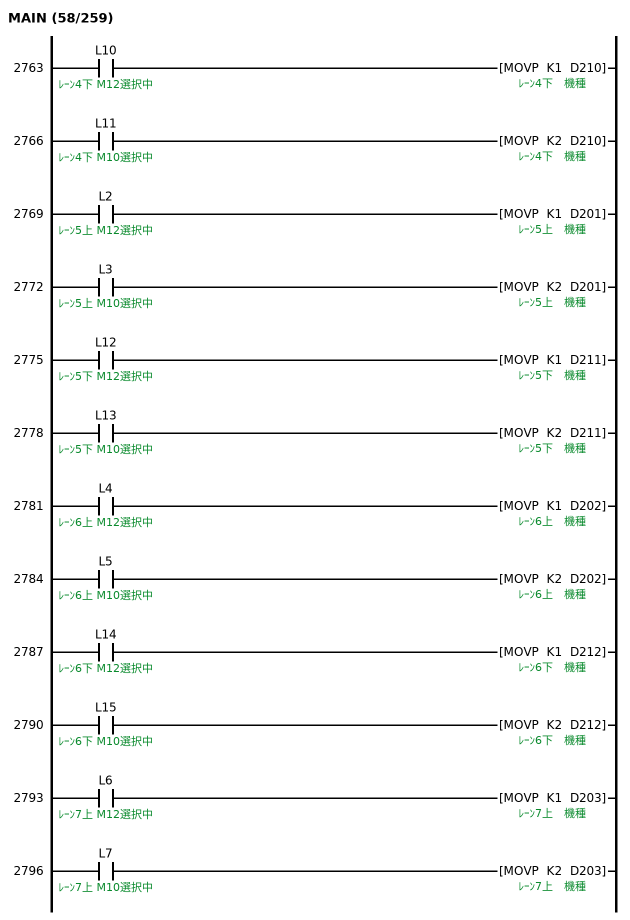
2763  LD      L10  ; ﾚｰﾝ4下 M12選択中
      MOVP    K1 D210  ; ﾚｰﾝ4下　機種
2766  LD      L11  ; ﾚｰﾝ4下 M10選択中
      MOVP    K2 D210
2769  LD      L2  ; ﾚｰﾝ5上 M12選択中
      MOVP    K1 D201  ; ﾚｰﾝ5上　機種
2772  LD      L3  ; ﾚｰﾝ5上 M10選択中
      MOVP    K2 D201
2775  LD      L12  ; ﾚｰﾝ5下 M12選択中
      MOVP    K1 D211  ; ﾚｰﾝ5下　機種
2778  LD      L13  ; ﾚｰﾝ5下 M10選択中
      MOVP    K2 D211
2781  LD      L4  ; ﾚｰﾝ6上 M12選択中
      MOVP    K1 D202  ; ﾚｰﾝ6上　機種
2784  LD      L5  ; ﾚｰﾝ6上 M10選択中
      MOVP    K2 D202
2787  LD      L14  ; ﾚｰﾝ6下 M12選択中
      MOVP    K1 D212  ; ﾚｰﾝ6下　機種
2790  LD      L15  ; ﾚｰﾝ6下 M10選択中
      MOVP    K2 D212
2793  LD      L6  ; ﾚｰﾝ7上 M12選択中
      MOVP    K1 D203  ; ﾚｰﾝ7上　機種
2796  LD      L7  ; ﾚｰﾝ7上 M10選択中
      MOVP    K2 D203
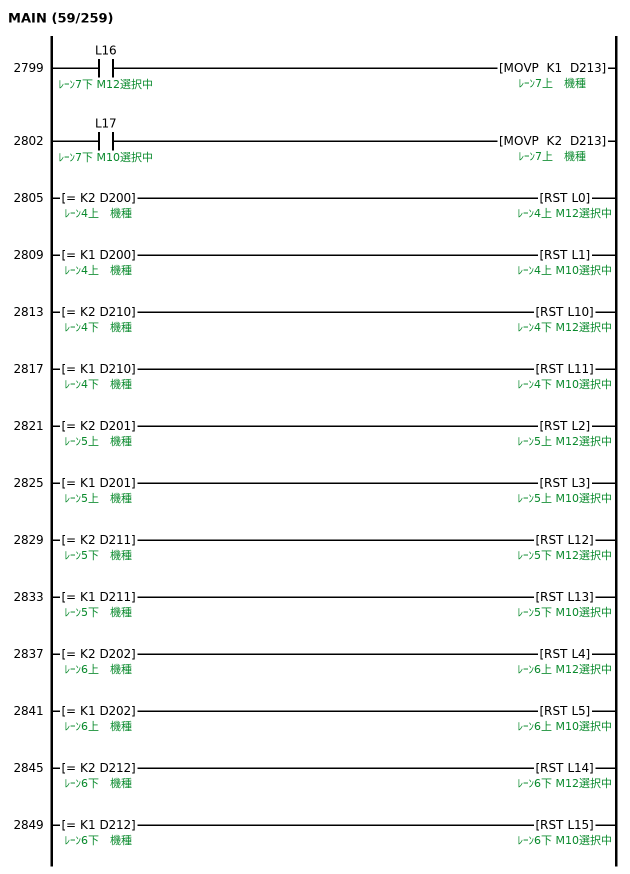
2799  LD      L16  ; ﾚｰﾝ7下 M12選択中
      MOVP    K1 D213  ; ﾚｰﾝ7上　機種
2802  LD      L17  ; ﾚｰﾝ7下 M10選択中
      MOVP    K2 D213
2805  LD=     K2 D200  ; ﾚｰﾝ4上　機種
      RST     L0  ; ﾚｰﾝ4上 M12選択中
2809  LD=     K1 D200  ; ﾚｰﾝ4上　機種
      RST     L1  ; ﾚｰﾝ4上 M10選択中
2813  LD=     K2 D210  ; ﾚｰﾝ4下　機種
      RST     L10  ; ﾚｰﾝ4下 M12選択中
2817  LD=     K1 D210  ; ﾚｰﾝ4下　機種
      RST     L11  ; ﾚｰﾝ4下 M10選択中
2821  LD=     K2 D201  ; ﾚｰﾝ5上　機種
      RST     L2  ; ﾚｰﾝ5上 M12選択中
2825  LD=     K1 D201  ; ﾚｰﾝ5上　機種
      RST     L3  ; ﾚｰﾝ5上 M10選択中
2829  LD=     K2 D211  ; ﾚｰﾝ5下　機種
      RST     L12  ; ﾚｰﾝ5下 M12選択中
2833  LD=     K1 D211  ; ﾚｰﾝ5下　機種
      RST     L13  ; ﾚｰﾝ5下 M10選択中
2837  LD=     K2 D202  ; ﾚｰﾝ6上　機種
      RST     L4  ; ﾚｰﾝ6上 M12選択中
2841  LD=     K1 D202  ; ﾚｰﾝ6上　機種
      RST     L5  ; ﾚｰﾝ6上 M10選択中
2845  LD=     K2 D212  ; ﾚｰﾝ6下　機種
      RST     L14  ; ﾚｰﾝ6下 M12選択中
2849  LD=     K1 D212  ; ﾚｰﾝ6下　機種
      RST     L15  ; ﾚｰﾝ6下 M10選択中
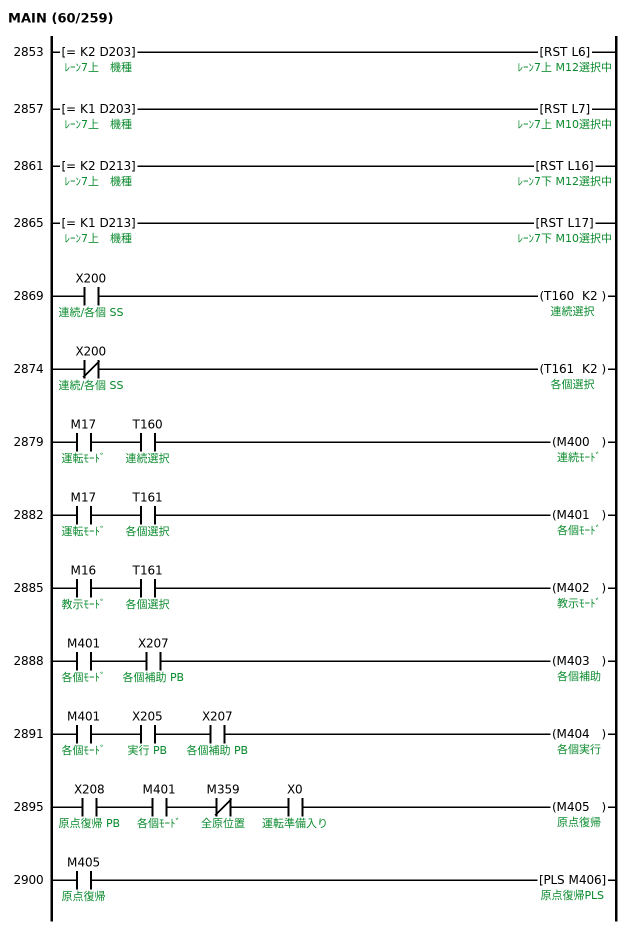
2853  LD=     K2 D203  ; ﾚｰﾝ7上　機種
      RST     L6  ; ﾚｰﾝ7上 M12選択中
2857  LD=     K1 D203  ; ﾚｰﾝ7上　機種
      RST     L7  ; ﾚｰﾝ7上 M10選択中
2861  LD=     K2 D213  ; ﾚｰﾝ7上　機種
      RST     L16  ; ﾚｰﾝ7下 M12選択中
2865  LD=     K1 D213  ; ﾚｰﾝ7上　機種
      RST     L17  ; ﾚｰﾝ7下 M10選択中
2869  LD      X200  ; 連続/各個 SS
      OUT     T160 K2  ; 連続選択
2874  LDI     X200  ; 連続/各個 SS
      OUT     T161 K2  ; 各個選択
2879  LD      M17  ; 運転ﾓｰﾄﾞ
      AND     T160  ; 連続選択
      OUT     M400  ; 連続ﾓｰﾄﾞ
2882  LD      M17  ; 運転ﾓｰﾄﾞ
      AND     T161  ; 各個選択
      OUT     M401  ; 各個ﾓｰﾄﾞ
2885  LD      M16  ; 教示ﾓｰﾄﾞ
      AND     T161  ; 各個選択
      OUT     M402  ; 教示ﾓｰﾄﾞ
2888  LD      M401  ; 各個ﾓｰﾄﾞ
      AND     X207  ; 各個補助 PB
      OUT     M403  ; 各個補助
2891  LD      M401  ; 各個ﾓｰﾄﾞ
      AND     X205  ; 実行 PB
      AND     X207  ; 各個補助 PB
      OUT     M404  ; 各個実行
2895  LD      X208  ; 原点復帰 PB
      AND     M401  ; 各個ﾓｰﾄﾞ
      ANI     M359  ; 全原位置
      AND     X0  ; 運転準備入り
      OUT     M405  ; 原点復帰
2900  LD      M405  ; 原点復帰
      PLS     M406  ; 原点復帰PLS
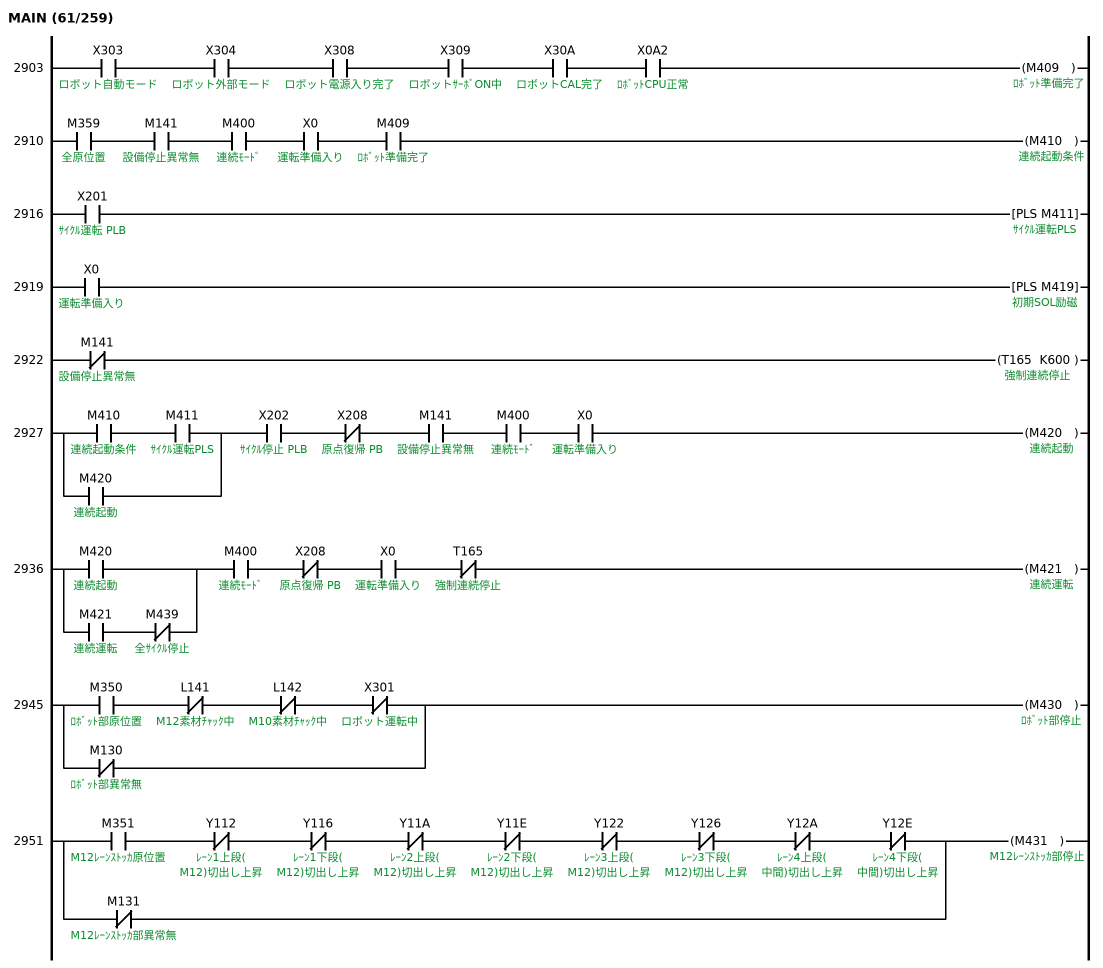
2903  LD      X303  ; ロボット自動モード
      AND     X304  ; ロボット外部モード
      AND     X308  ; ロボット電源入り完了
      AND     X309  ; ロボットｻｰﾎﾞON中
      AND     X30A  ; ロボットCAL完了
      AND     X0A2  ; ﾛﾎﾞｯﾄCPU正常
      OUT     M409  ; ﾛﾎﾞｯﾄ準備完了
2910  LD      M359  ; 全原位置
      AND     M141  ; 設備停止異常無
      AND     M400  ; 連続ﾓｰﾄﾞ
      AND     X0  ; 運転準備入り
      AND     M409  ; ﾛﾎﾞｯﾄ準備完了
      OUT     M410  ; 連続起動条件
2916  LD      X201  ; ｻｲｸﾙ運転 PLB
      PLS     M411  ; ｻｲｸﾙ運転PLS
2919  LD      X0  ; 運転準備入り
      PLS     M419  ; 初期SOL励磁
2922  LDI     M141  ; 設備停止異常無
      OUT     T165 K600  ; 強制連続停止
2927  LD      M410  ; 連続起動条件
      AND     M411  ; ｻｲｸﾙ運転PLS
      OR      M420  ; 連続起動
      AND     X202  ; ｻｲｸﾙ停止 PLB
      ANI     X208  ; 原点復帰 PB
      AND     M141  ; 設備停止異常無
      AND     M400  ; 連続ﾓｰﾄﾞ
      AND     X0  ; 運転準備入り
      OUT     M420  ; 連続起動
2936  LD      M420  ; 連続起動
      LD      M421  ; 連続運転
      ANI     M439  ; 全ｻｲｸﾙ停止
      ORB
      AND     M400  ; 連続ﾓｰﾄﾞ
      ANI     X208  ; 原点復帰 PB
      AND     X0  ; 運転準備入り
      ANI     T165  ; 強制連続停止
      OUT     M421  ; 連続運転
2945  LD      M350  ; ﾛﾎﾞｯﾄ部原位置
      ANI     L141  ; M12素材ﾁｬｯｸ中
      ANI     L142  ; M10素材ﾁｬｯｸ中
      ANI     X301  ; ロボット運転中
      ORI     M130  ; ﾛﾎﾞｯﾄ部異常無
      OUT     M430  ; ﾛﾎﾞｯﾄ部停止
2951  LD      M351  ; M12ﾚｰﾝｽﾄｯｶ原位置
      ANI     Y112  ; ﾚｰﾝ1上段(M12)切出し上昇
      ANI     Y116  ; ﾚｰﾝ1下段(M12)切出し上昇
      ANI     Y11A  ; ﾚｰﾝ2上段(M12)切出し上昇
      ANI     Y11E  ; ﾚｰﾝ2下段(M12)切出し上昇
      ANI     Y122  ; ﾚｰﾝ3上段(M12)切出し上昇
      ANI     Y126  ; ﾚｰﾝ3下段(M12)切出し上昇
      ANI     Y12A  ; ﾚｰﾝ4上段(中間)切出し上昇
      ANI     Y12E  ; ﾚｰﾝ4下段(中間)切出し上昇
      ORI     M131  ; M12ﾚｰﾝｽﾄｯｶ部異常無
      OUT     M431  ; M12ﾚｰﾝｽﾄｯｶ部停止
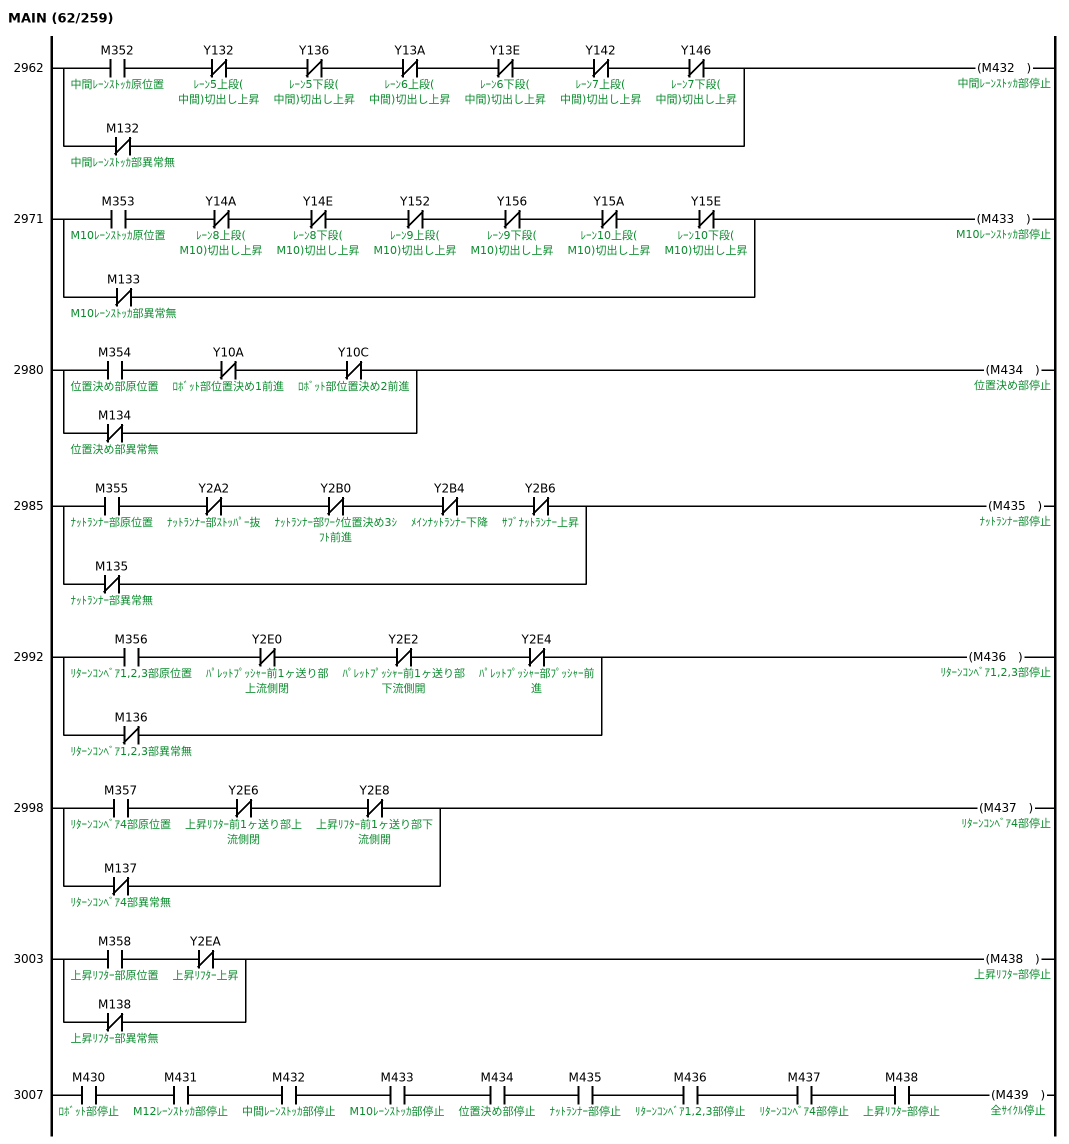
2962  LD      M352  ; 中間ﾚｰﾝｽﾄｯｶ原位置
      ANI     Y132  ; ﾚｰﾝ5上段(中間)切出し上昇
      ANI     Y136  ; ﾚｰﾝ5下段(中間)切出し上昇
      ANI     Y13A  ; ﾚｰﾝ6上段(中間)切出し上昇
      ANI     Y13E  ; ﾚｰﾝ6下段(中間)切出し上昇
      ANI     Y142  ; ﾚｰﾝ7上段(中間)切出し上昇
      ANI     Y146  ; ﾚｰﾝ7下段(中間)切出し上昇
      ORI     M132  ; 中間ﾚｰﾝｽﾄｯｶ部異常無
      OUT     M432  ; 中間ﾚｰﾝｽﾄｯｶ部停止
2971  LD      M353  ; M10ﾚｰﾝｽﾄｯｶ原位置
      ANI     Y14A  ; ﾚｰﾝ8上段(M10)切出し上昇
      ANI     Y14E  ; ﾚｰﾝ8下段(M10)切出し上昇
      ANI     Y152  ; ﾚｰﾝ9上段(M10)切出し上昇
      ANI     Y156  ; ﾚｰﾝ9下段(M10)切出し上昇
      ANI     Y15A  ; ﾚｰﾝ10上段(M10)切出し上昇
      ANI     Y15E  ; ﾚｰﾝ10下段(M10)切出し上昇
      ORI     M133  ; M10ﾚｰﾝｽﾄｯｶ部異常無
      OUT     M433  ; M10ﾚｰﾝｽﾄｯｶ部停止
2980  LD      M354  ; 位置決め部原位置
      ANI     Y10A  ; ﾛﾎﾞｯﾄ部位置決め1前進
      ANI     Y10C  ; ﾛﾎﾞｯﾄ部位置決め2前進
      ORI     M134  ; 位置決め部異常無
      OUT     M434  ; 位置決め部停止
2985  LD      M355  ; ﾅｯﾄﾗﾝﾅｰ部原位置
      ANI     Y2A2  ; ﾅｯﾄﾗﾝﾅｰ部ｽﾄｯﾊﾟｰ抜
      ANI     Y2B0  ; ﾅｯﾄﾗﾝﾅｰ部ﾜｰｸ位置決め3ｼﾌﾄ前進
      ANI     Y2B4  ; ﾒｲﾝﾅｯﾄﾗﾝﾅｰ下降
      ANI     Y2B6  ; ｻﾌﾞﾅｯﾄﾗﾝﾅｰ上昇
      ORI     M135  ; ﾅｯﾄﾗﾝﾅｰ部異常無
      OUT     M435  ; ﾅｯﾄﾗﾝﾅｰ部停止
2992  LD      M356  ; ﾘﾀｰﾝｺﾝﾍﾞｱ1,2,3部原位置
      ANI     Y2E0  ; ﾊﾟﾚｯﾄﾌﾟｯｼｬｰ前1ヶ送り部上流側閉
      ANI     Y2E2  ; ﾊﾟﾚｯﾄﾌﾟｯｼｬｰ前1ヶ送り部下流側開
      ANI     Y2E4  ; ﾊﾟﾚｯﾄﾌﾟｯｼｬｰ部ﾌﾟｯｼｬｰ前進
      ORI     M136  ; ﾘﾀｰﾝｺﾝﾍﾞｱ1,2,3部異常無
      OUT     M436  ; ﾘﾀｰﾝｺﾝﾍﾞｱ1,2,3部停止
2998  LD      M357  ; ﾘﾀｰﾝｺﾝﾍﾞｱ4部原位置
      ANI     Y2E6  ; 上昇ﾘﾌﾀｰ前1ヶ送り部上流側閉
      ANI     Y2E8  ; 上昇ﾘﾌﾀｰ前1ヶ送り部下流側開
      ORI     M137  ; ﾘﾀｰﾝｺﾝﾍﾞｱ4部異常無
      OUT     M437  ; ﾘﾀｰﾝｺﾝﾍﾞｱ4部停止
3003  LD      M358  ; 上昇ﾘﾌﾀｰ部原位置
      ANI     Y2EA  ; 上昇ﾘﾌﾀｰ上昇
      ORI     M138  ; 上昇ﾘﾌﾀｰ部異常無
      OUT     M438  ; 上昇ﾘﾌﾀｰ部停止
3007  LD      M430  ; ﾛﾎﾞｯﾄ部停止
      AND     M431  ; M12ﾚｰﾝｽﾄｯｶ部停止
      AND     M432  ; 中間ﾚｰﾝｽﾄｯｶ部停止
      AND     M433  ; M10ﾚｰﾝｽﾄｯｶ部停止
      AND     M434  ; 位置決め部停止
      AND     M435  ; ﾅｯﾄﾗﾝﾅｰ部停止
      AND     M436  ; ﾘﾀｰﾝｺﾝﾍﾞｱ1,2,3部停止
      AND     M437  ; ﾘﾀｰﾝｺﾝﾍﾞｱ4部停止
      AND     M438  ; 上昇ﾘﾌﾀｰ部停止
      OUT     M439  ; 全ｻｲｸﾙ停止
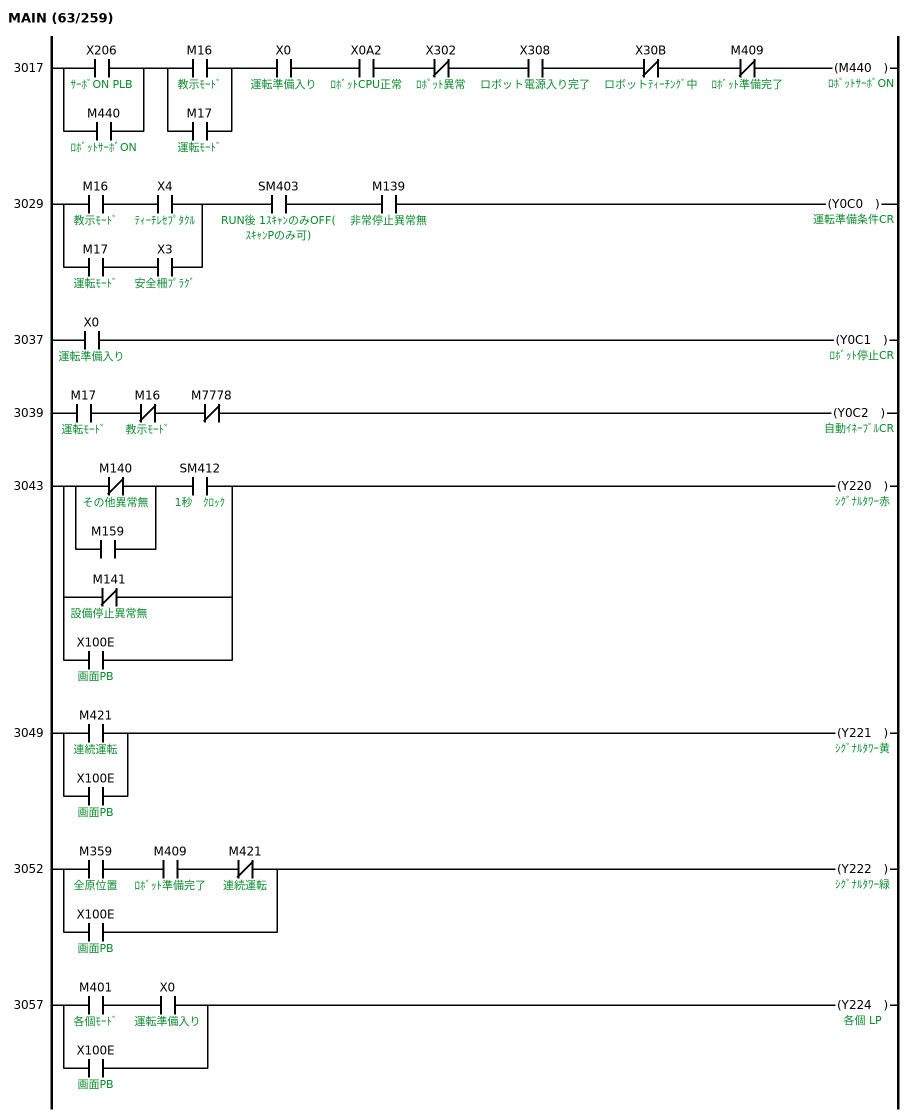
3017  LD      X206  ; ｻｰﾎﾞON PLB
      OR      M440  ; ﾛﾎﾞｯﾄｻｰﾎﾞON
      LD      M16  ; 教示ﾓｰﾄﾞ
      OR      M17  ; 運転ﾓｰﾄﾞ
      ANB
      AND     X0  ; 運転準備入り
      AND     X0A2  ; ﾛﾎﾞｯﾄCPU正常
      ANI     X302  ; ﾛﾎﾞｯﾄ異常
      AND     X308  ; ロボット電源入り完了
      ANI     X30B  ; ロボットﾃｨｰﾁﾝｸﾞ中
      ANI     M409  ; ﾛﾎﾞｯﾄ準備完了
      OUT     M440  ; ﾛﾎﾞｯﾄｻｰﾎﾞON
3029  LD      M16  ; 教示ﾓｰﾄﾞ
      AND     X4  ; ﾃｨｰﾁﾚｾﾌﾟﾀｸﾙ
      LD      M17  ; 運転ﾓｰﾄﾞ
      AND     X3  ; 安全柵ﾌﾟﾗｸﾞ
      ORB
      AND     SM403  ; RUN後 1ｽｷｬﾝのみOFF(ｽｷｬﾝPのみ可)
      AND     M139  ; 非常停止異常無
      OUT     Y0C0  ; 運転準備条件CR
3037  LD      X0  ; 運転準備入り
      OUT     Y0C1  ; ﾛﾎﾞｯﾄ停止CR
3039  LD      M17  ; 運転ﾓｰﾄﾞ
      ANI     M16  ; 教示ﾓｰﾄﾞ
      ANI     M7778
      OUT     Y0C2  ; 自動ｲﾈｰﾌﾞﾙCR
3043  LDI     M140  ; その他異常無
      OR      M159
      AND     SM412  ; 1秒   ｸﾛｯｸ
      ORI     M141  ; 設備停止異常無
      OR      X100E  ; 画面PB
      OUT     Y220  ; ｼｸﾞﾅﾙﾀﾜｰ赤
3049  LD      M421  ; 連続運転
      OR      X100E  ; 画面PB
      OUT     Y221  ; ｼｸﾞﾅﾙﾀﾜｰ黄
3052  LD      M359  ; 全原位置
      AND     M409  ; ﾛﾎﾞｯﾄ準備完了
      ANI     M421  ; 連続運転
      OR      X100E  ; 画面PB
      OUT     Y222  ; ｼｸﾞﾅﾙﾀﾜｰ緑
3057  LD      M401  ; 各個ﾓｰﾄﾞ
      AND     X0  ; 運転準備入り
      OR      X100E  ; 画面PB
      OUT     Y224  ; 各個 LP
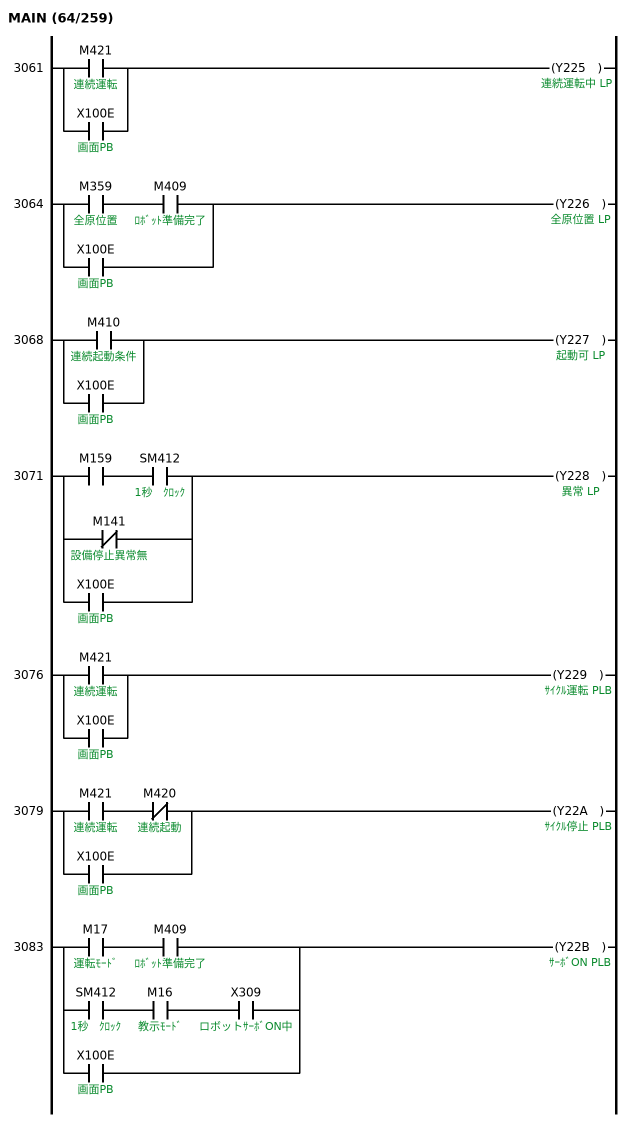
3061  LD      M421  ; 連続運転
      OR      X100E  ; 画面PB
      OUT     Y225  ; 連続運転中 LP
3064  LD      M359  ; 全原位置
      AND     M409  ; ﾛﾎﾞｯﾄ準備完了
      OR      X100E  ; 画面PB
      OUT     Y226  ; 全原位置 LP
3068  LD      M410  ; 連続起動条件
      OR      X100E  ; 画面PB
      OUT     Y227  ; 起動可 LP
3071  LD      M159
      AND     SM412  ; 1秒   ｸﾛｯｸ
      ORI     M141  ; 設備停止異常無
      OR      X100E  ; 画面PB
      OUT     Y228  ; 異常 LP
3076  LD      M421  ; 連続運転
      OR      X100E  ; 画面PB
      OUT     Y229  ; ｻｲｸﾙ運転 PLB
3079  LD      M421  ; 連続運転
      ANI     M420  ; 連続起動
      OR      X100E  ; 画面PB
      OUT     Y22A  ; ｻｲｸﾙ停止 PLB
3083  LD      M17  ; 運転ﾓｰﾄﾞ
      AND     M409  ; ﾛﾎﾞｯﾄ準備完了
      LD      SM412  ; 1秒   ｸﾛｯｸ
      AND     M16  ; 教示ﾓｰﾄﾞ
      AND     X309  ; ロボットｻｰﾎﾞON中
      ORB
      OR      X100E  ; 画面PB
      OUT     Y22B  ; ｻｰﾎﾞON PLB
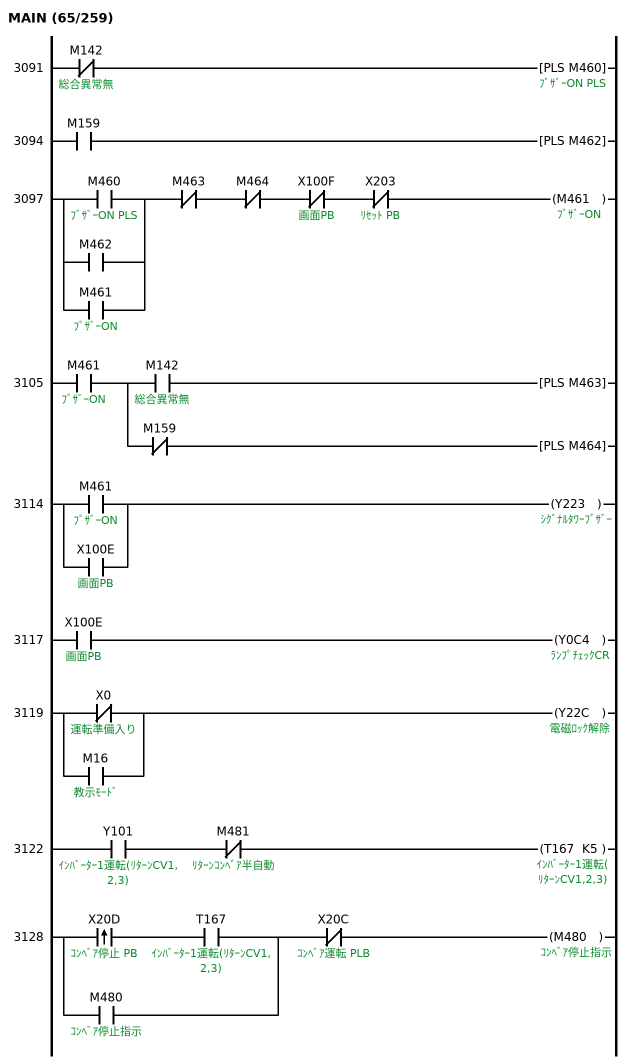
3091  LDI     M142  ; 総合異常無
      PLS     M460  ; ﾌﾞｻﾞｰON PLS
3094  LD      M159
      PLS     M462
3097  LD      M460  ; ﾌﾞｻﾞｰON PLS
      OR      M462
      OR      M461  ; ﾌﾞｻﾞｰON
      ANI     M463
      ANI     M464
      ANI     X100F  ; 画面PB
      ANI     X203  ; ﾘｾｯﾄ PB
      OUT     M461  ; ﾌﾞｻﾞｰON
3105  LD      M461  ; ﾌﾞｻﾞｰON
      MPS
      AND     M142  ; 総合異常無
      PLS     M463
      MPP
      ANI     M159
      PLS     M464
3114  LD      M461  ; ﾌﾞｻﾞｰON
      OR      X100E  ; 画面PB
      OUT     Y223  ; ｼｸﾞﾅﾙﾀﾜｰﾌﾞｻﾞｰ
3117  LD      X100E  ; 画面PB
      OUT     Y0C4  ; ﾗﾝﾌﾟﾁｪｯｸCR
3119  LDI     X0  ; 運転準備入り
      OR      M16  ; 教示ﾓｰﾄﾞ
      OUT     Y22C  ; 電磁ﾛｯｸ解除
3122  LD      Y101  ; ｲﾝﾊﾞｰﾀｰ1運転(ﾘﾀｰﾝCV1,2,3)
      ANI     M481  ; ﾘﾀｰﾝｺﾝﾍﾞｱ半自動
      OUT     T167 K5  ; ｲﾝﾊﾞｰﾀｰ1運転(ﾘﾀｰﾝCV1,2,3)
3128  LDP     X20D  ; ｺﾝﾍﾞｱ停止 PB
      AND     T167  ; ｲﾝﾊﾞｰﾀｰ1運転(ﾘﾀｰﾝCV1,2,3)
      OR      M480  ; ｺﾝﾍﾞｱ停止指示
      ANI     X20C  ; ｺﾝﾍﾞｱ運転 PLB
      OUT     M480  ; ｺﾝﾍﾞｱ停止指示
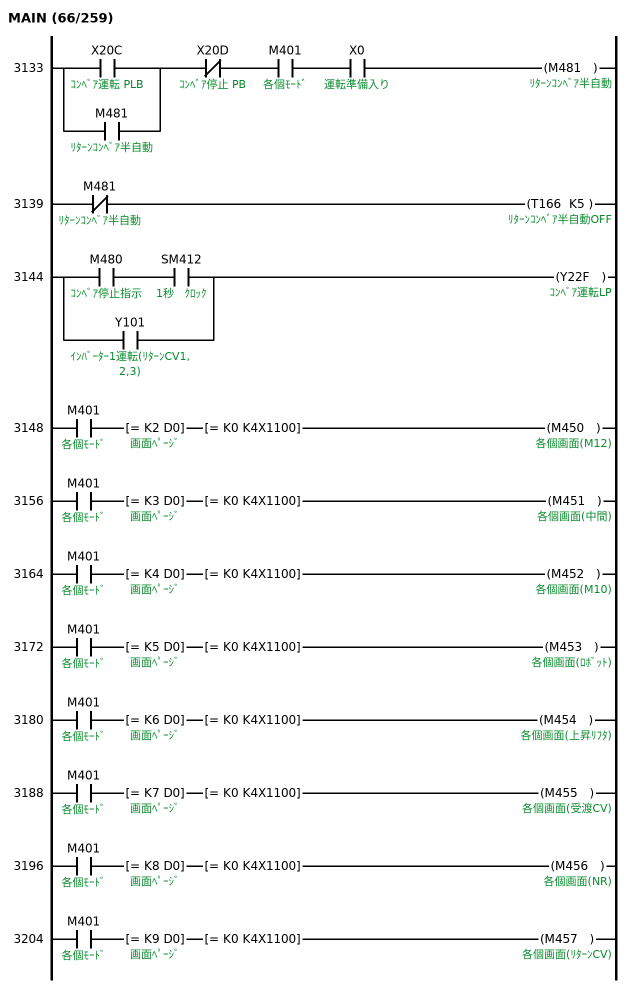
3133  LD      X20C  ; ｺﾝﾍﾞｱ運転 PLB
      OR      M481  ; ﾘﾀｰﾝｺﾝﾍﾞｱ半自動
      ANI     X20D  ; ｺﾝﾍﾞｱ停止 PB
      AND     M401  ; 各個ﾓｰﾄﾞ
      AND     X0  ; 運転準備入り
      OUT     M481  ; ﾘﾀｰﾝｺﾝﾍﾞｱ半自動
3139  LDI     M481  ; ﾘﾀｰﾝｺﾝﾍﾞｱ半自動
      OUT     T166 K5  ; ﾘﾀｰﾝｺﾝﾍﾞｱ半自動OFF
3144  LD      M480  ; ｺﾝﾍﾞｱ停止指示
      AND     SM412  ; 1秒   ｸﾛｯｸ
      OR      Y101  ; ｲﾝﾊﾞｰﾀｰ1運転(ﾘﾀｰﾝCV1,2,3)
      OUT     Y22F  ; ｺﾝﾍﾞｱ運転LP
3148  LD      M401  ; 各個ﾓｰﾄﾞ
      AND=    K2 D0  ; 画面ﾍﾟｰｼﾞ
      AND=    K0 K4X1100  ; 画面PLB
      OUT     M450  ; 各個画面(M12)
3156  LD      M401  ; 各個ﾓｰﾄﾞ
      AND=    K3 D0  ; 画面ﾍﾟｰｼﾞ
      AND=    K0 K4X1100  ; 画面PLB
      OUT     M451  ; 各個画面(中間)
3164  LD      M401  ; 各個ﾓｰﾄﾞ
      AND=    K4 D0  ; 画面ﾍﾟｰｼﾞ
      AND=    K0 K4X1100  ; 画面PLB
      OUT     M452  ; 各個画面(M10)
3172  LD      M401  ; 各個ﾓｰﾄﾞ
      AND=    K5 D0  ; 画面ﾍﾟｰｼﾞ
      AND=    K0 K4X1100  ; 画面PLB
      OUT     M453  ; 各個画面(ﾛﾎﾞｯﾄ)
3180  LD      M401  ; 各個ﾓｰﾄﾞ
      AND=    K6 D0  ; 画面ﾍﾟｰｼﾞ
      AND=    K0 K4X1100  ; 画面PLB
      OUT     M454  ; 各個画面(上昇ﾘﾌﾀ)
3188  LD      M401  ; 各個ﾓｰﾄﾞ
      AND=    K7 D0  ; 画面ﾍﾟｰｼﾞ
      AND=    K0 K4X1100  ; 画面PLB
      OUT     M455  ; 各個画面(受渡CV)
3196  LD      M401  ; 各個ﾓｰﾄﾞ
      AND=    K8 D0  ; 画面ﾍﾟｰｼﾞ
      AND=    K0 K4X1100  ; 画面PLB
      OUT     M456  ; 各個画面(NR)
3204  LD      M401  ; 各個ﾓｰﾄﾞ
      AND=    K9 D0  ; 画面ﾍﾟｰｼﾞ
      AND=    K0 K4X1100  ; 画面PLB
      OUT     M457  ; 各個画面(ﾘﾀｰﾝCV)
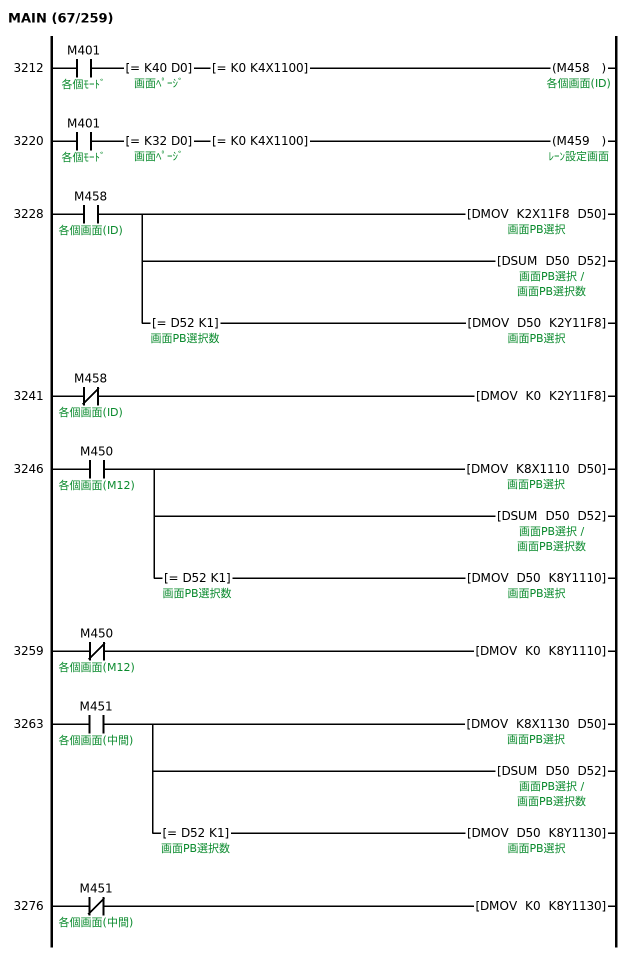
3212  LD      M401  ; 各個ﾓｰﾄﾞ
      AND=    K40 D0  ; 画面ﾍﾟｰｼﾞ
      AND=    K0 K4X1100  ; 画面PLB
      OUT     M458  ; 各個画面(ID)
3220  LD      M401  ; 各個ﾓｰﾄﾞ
      AND=    K32 D0  ; 画面ﾍﾟｰｼﾞ
      AND=    K0 K4X1100  ; 画面PLB
      OUT     M459  ; ﾚｰﾝ設定画面
3228  LD      M458  ; 各個画面(ID)
      DMOV    K2X11F8 D50  ; 画面PLB / 画面PB選択
      DSUM    D50 D52  ; 画面PB選択数
      AND=    D52 K1  ; 画面PB選択数
      DMOV    D50 K2Y11F8  ; 画面PLB
3241  LDI     M458  ; 各個画面(ID)
      DMOV    K0 K2Y11F8
3246  LD      M450  ; 各個画面(M12)
      DMOV    K8X1110 D50  ; 画面PLB
      DSUM    D50 D52
      AND=    D52 K1  ; 画面PB選択数
      DMOV    D50 K8Y1110  ; 画面PLB
3259  LDI     M450  ; 各個画面(M12)
      DMOV    K0 K8Y1110
3263  LD      M451  ; 各個画面(中間)
      DMOV    K8X1130 D50  ; 画面PLB
      DSUM    D50 D52
      AND=    D52 K1  ; 画面PB選択数
      DMOV    D50 K8Y1130  ; 画面PLB
3276  LDI     M451  ; 各個画面(中間)
      DMOV    K0 K8Y1130
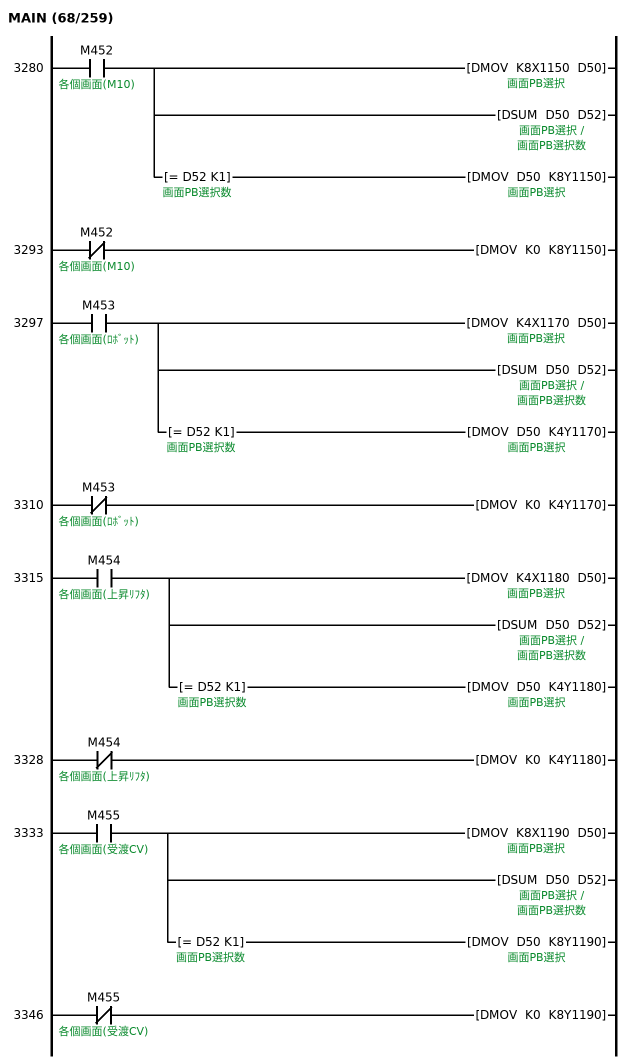
3280  LD      M452  ; 各個画面(M10)
      DMOV    K8X1150 D50  ; 画面PLB
      DSUM    D50 D52
      AND=    D52 K1  ; 画面PB選択数
      DMOV    D50 K8Y1150  ; 画面PLB
3293  LDI     M452  ; 各個画面(M10)
      DMOV    K0 K8Y1150
3297  LD      M453  ; 各個画面(ﾛﾎﾞｯﾄ)
      DMOV    K4X1170 D50  ; 画面PLB
      DSUM    D50 D52
      AND=    D52 K1  ; 画面PB選択数
      DMOV    D50 K4Y1170  ; 画面PLB
3310  LDI     M453  ; 各個画面(ﾛﾎﾞｯﾄ)
      DMOV    K0 K4Y1170
3315  LD      M454  ; 各個画面(上昇ﾘﾌﾀ)
      DMOV    K4X1180 D50  ; 画面PLB
      DSUM    D50 D52
      AND=    D52 K1  ; 画面PB選択数
      DMOV    D50 K4Y1180  ; 画面PLB
3328  LDI     M454  ; 各個画面(上昇ﾘﾌﾀ)
      DMOV    K0 K4Y1180
3333  LD      M455  ; 各個画面(受渡CV)
      DMOV    K8X1190 D50  ; 画面PLB
      DSUM    D50 D52
      AND=    D52 K1  ; 画面PB選択数
      DMOV    D50 K8Y1190  ; 画面PLB
3346  LDI     M455  ; 各個画面(受渡CV)
      DMOV    K0 K8Y1190
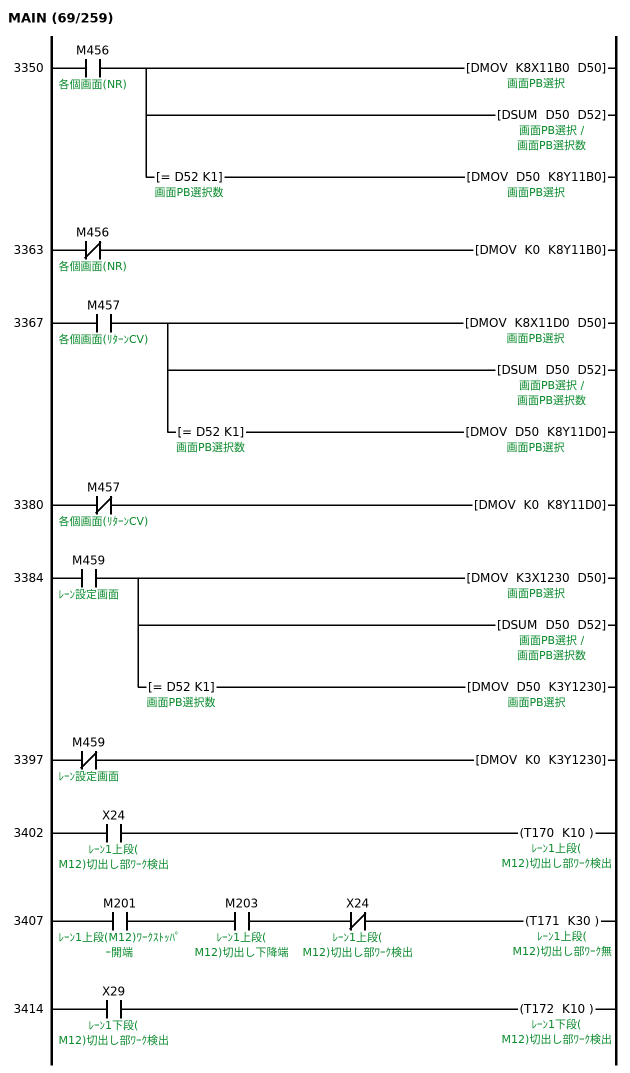
3350  LD      M456  ; 各個画面(NR)
      DMOV    K8X11B0 D50  ; 画面PLB
      DSUM    D50 D52
      AND=    D52 K1  ; 画面PB選択数
      DMOV    D50 K8Y11B0  ; 画面PLB
3363  LDI     M456  ; 各個画面(NR)
      DMOV    K0 K8Y11B0
3367  LD      M457  ; 各個画面(ﾘﾀｰﾝCV)
      DMOV    K8X11D0 D50  ; 画面PLB
      DSUM    D50 D52
      AND=    D52 K1  ; 画面PB選択数
      DMOV    D50 K8Y11D0  ; 画面PLB
3380  LDI     M457  ; 各個画面(ﾘﾀｰﾝCV)
      DMOV    K0 K8Y11D0
3384  LD      M459  ; ﾚｰﾝ設定画面
      DMOV    K3X1230 D50  ; 画面PLB
      DSUM    D50 D52
      AND=    D52 K1  ; 画面PB選択数
      DMOV    D50 K3Y1230
3397  LDI     M459  ; ﾚｰﾝ設定画面
      DMOV    K0 K3Y1230
3402  LD      X24  ; ﾚｰﾝ1上段(M12)切出し部ﾜｰｸ検出
      OUT     T170 K10  ; ﾚｰﾝ1上段(M12)切出し部ﾜｰｸ検出
3407  LD      M201  ; ﾚｰﾝ1上段(M12)ﾜｰｸｽﾄｯﾊﾟｰ開端
      AND     M203  ; ﾚｰﾝ1上段(M12)切出し下降端
      ANI     X24  ; ﾚｰﾝ1上段(M12)切出し部ﾜｰｸ検出
      OUT     T171 K30  ; ﾚｰﾝ1上段(M12)切出し部ﾜｰｸ無
3414  LD      X29  ; ﾚｰﾝ1下段(M12)切出し部ﾜｰｸ検出
      OUT     T172 K10  ; ﾚｰﾝ1下段(M12)切出し部ﾜｰｸ検出
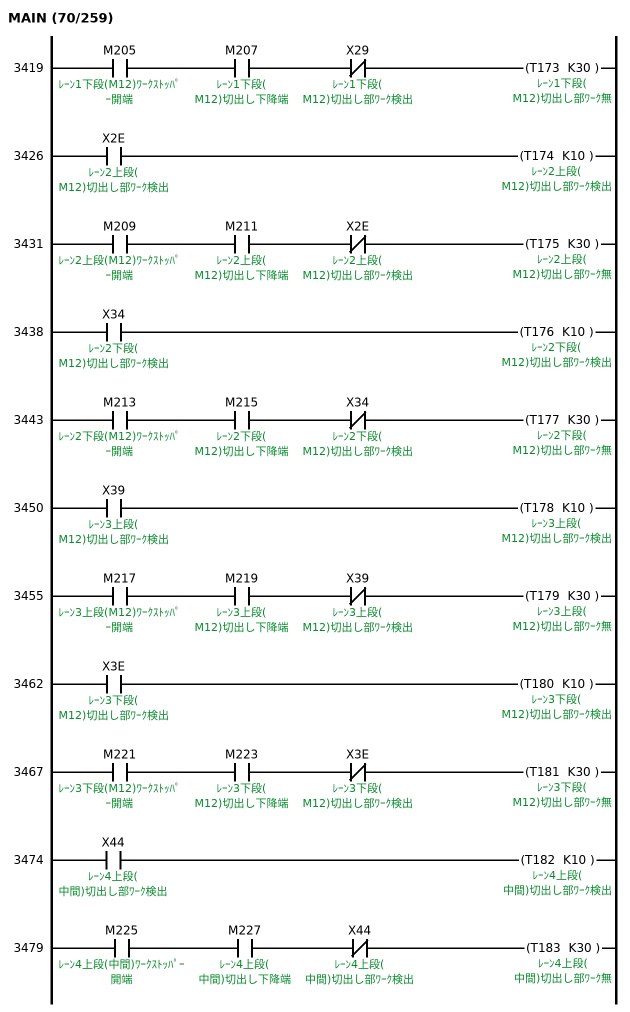
3419  LD      M205  ; ﾚｰﾝ1下段(M12)ﾜｰｸｽﾄｯﾊﾟｰ開端
      AND     M207  ; ﾚｰﾝ1下段(M12)切出し下降端
      ANI     X29  ; ﾚｰﾝ1下段(M12)切出し部ﾜｰｸ検出
      OUT     T173 K30  ; ﾚｰﾝ1下段(M12)切出し部ﾜｰｸ無
3426  LD      X2E  ; ﾚｰﾝ2上段(M12)切出し部ﾜｰｸ検出
      OUT     T174 K10  ; ﾚｰﾝ2上段(M12)切出し部ﾜｰｸ検出
3431  LD      M209  ; ﾚｰﾝ2上段(M12)ﾜｰｸｽﾄｯﾊﾟｰ開端
      AND     M211  ; ﾚｰﾝ2上段(M12)切出し下降端
      ANI     X2E  ; ﾚｰﾝ2上段(M12)切出し部ﾜｰｸ検出
      OUT     T175 K30  ; ﾚｰﾝ2上段(M12)切出し部ﾜｰｸ無
3438  LD      X34  ; ﾚｰﾝ2下段(M12)切出し部ﾜｰｸ検出
      OUT     T176 K10  ; ﾚｰﾝ2下段(M12)切出し部ﾜｰｸ検出
3443  LD      M213  ; ﾚｰﾝ2下段(M12)ﾜｰｸｽﾄｯﾊﾟｰ開端
      AND     M215  ; ﾚｰﾝ2下段(M12)切出し下降端
      ANI     X34  ; ﾚｰﾝ2下段(M12)切出し部ﾜｰｸ検出
      OUT     T177 K30  ; ﾚｰﾝ2下段(M12)切出し部ﾜｰｸ無
3450  LD      X39  ; ﾚｰﾝ3上段(M12)切出し部ﾜｰｸ検出
      OUT     T178 K10  ; ﾚｰﾝ3上段(M12)切出し部ﾜｰｸ検出
3455  LD      M217  ; ﾚｰﾝ3上段(M12)ﾜｰｸｽﾄｯﾊﾟｰ開端
      AND     M219  ; ﾚｰﾝ3上段(M12)切出し下降端
      ANI     X39  ; ﾚｰﾝ3上段(M12)切出し部ﾜｰｸ検出
      OUT     T179 K30  ; ﾚｰﾝ3上段(M12)切出し部ﾜｰｸ無
3462  LD      X3E  ; ﾚｰﾝ3下段(M12)切出し部ﾜｰｸ検出
      OUT     T180 K10  ; ﾚｰﾝ3下段(M12)切出し部ﾜｰｸ検出
3467  LD      M221  ; ﾚｰﾝ3下段(M12)ﾜｰｸｽﾄｯﾊﾟｰ開端
      AND     M223  ; ﾚｰﾝ3下段(M12)切出し下降端
      ANI     X3E  ; ﾚｰﾝ3下段(M12)切出し部ﾜｰｸ検出
      OUT     T181 K30  ; ﾚｰﾝ3下段(M12)切出し部ﾜｰｸ無
3474  LD      X44  ; ﾚｰﾝ4上段(中間)切出し部ﾜｰｸ検出
      OUT     T182 K10  ; ﾚｰﾝ4上段(中間)切出し部ﾜｰｸ検出
3479  LD      M225  ; ﾚｰﾝ4上段(中間)ﾜｰｸｽﾄｯﾊﾟｰ開端
      AND     M227  ; ﾚｰﾝ4上段(中間)切出し下降端
      ANI     X44  ; ﾚｰﾝ4上段(中間)切出し部ﾜｰｸ検出
      OUT     T183 K30  ; ﾚｰﾝ4上段(中間)切出し部ﾜｰｸ無
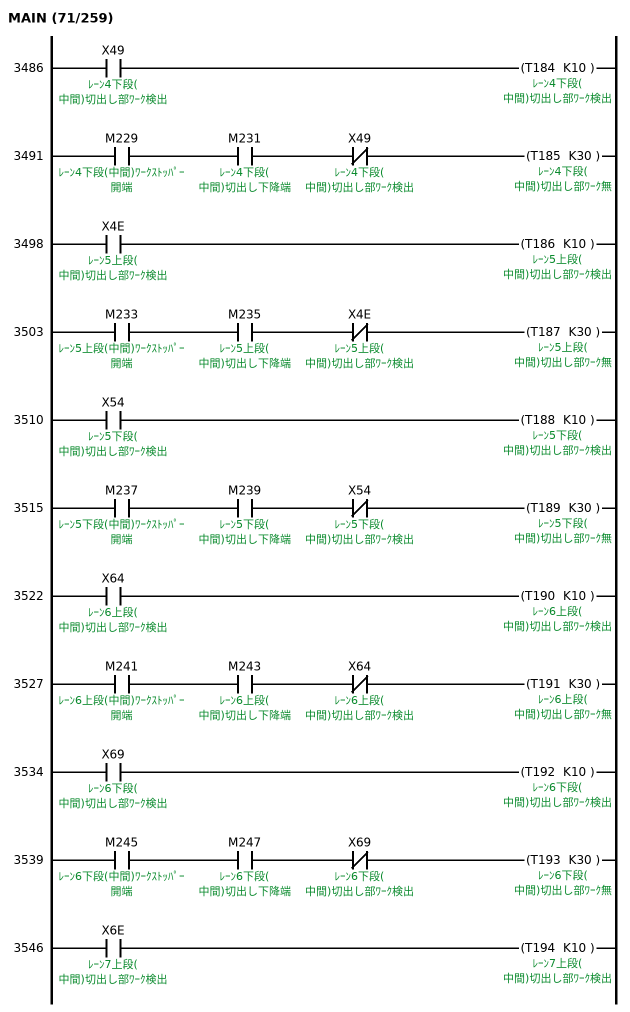
3486  LD      X49  ; ﾚｰﾝ4下段(中間)切出し部ﾜｰｸ検出
      OUT     T184 K10  ; ﾚｰﾝ4下段(中間)切出し部ﾜｰｸ検出
3491  LD      M229  ; ﾚｰﾝ4下段(中間)ﾜｰｸｽﾄｯﾊﾟｰ開端
      AND     M231  ; ﾚｰﾝ4下段(中間)切出し下降端
      ANI     X49  ; ﾚｰﾝ4下段(中間)切出し部ﾜｰｸ検出
      OUT     T185 K30  ; ﾚｰﾝ4下段(中間)切出し部ﾜｰｸ無
3498  LD      X4E  ; ﾚｰﾝ5上段(中間)切出し部ﾜｰｸ検出
      OUT     T186 K10  ; ﾚｰﾝ5上段(中間)切出し部ﾜｰｸ検出
3503  LD      M233  ; ﾚｰﾝ5上段(中間)ﾜｰｸｽﾄｯﾊﾟｰ開端
      AND     M235  ; ﾚｰﾝ5上段(中間)切出し下降端
      ANI     X4E  ; ﾚｰﾝ5上段(中間)切出し部ﾜｰｸ検出
      OUT     T187 K30  ; ﾚｰﾝ5上段(中間)切出し部ﾜｰｸ無
3510  LD      X54  ; ﾚｰﾝ5下段(中間)切出し部ﾜｰｸ検出
      OUT     T188 K10  ; ﾚｰﾝ5下段(中間)切出し部ﾜｰｸ検出
3515  LD      M237  ; ﾚｰﾝ5下段(中間)ﾜｰｸｽﾄｯﾊﾟｰ開端
      AND     M239  ; ﾚｰﾝ5下段(中間)切出し下降端
      ANI     X54  ; ﾚｰﾝ5下段(中間)切出し部ﾜｰｸ検出
      OUT     T189 K30  ; ﾚｰﾝ5下段(中間)切出し部ﾜｰｸ無
3522  LD      X64  ; ﾚｰﾝ6上段(中間)切出し部ﾜｰｸ検出
      OUT     T190 K10  ; ﾚｰﾝ6上段(中間)切出し部ﾜｰｸ検出
3527  LD      M241  ; ﾚｰﾝ6上段(中間)ﾜｰｸｽﾄｯﾊﾟｰ開端
      AND     M243  ; ﾚｰﾝ6上段(中間)切出し下降端
      ANI     X64  ; ﾚｰﾝ6上段(中間)切出し部ﾜｰｸ検出
      OUT     T191 K30  ; ﾚｰﾝ6上段(中間)切出し部ﾜｰｸ無
3534  LD      X69  ; ﾚｰﾝ6下段(中間)切出し部ﾜｰｸ検出
      OUT     T192 K10  ; ﾚｰﾝ6下段(中間)切出し部ﾜｰｸ検出
3539  LD      M245  ; ﾚｰﾝ6下段(中間)ﾜｰｸｽﾄｯﾊﾟｰ開端
      AND     M247  ; ﾚｰﾝ6下段(中間)切出し下降端
      ANI     X69  ; ﾚｰﾝ6下段(中間)切出し部ﾜｰｸ検出
      OUT     T193 K30  ; ﾚｰﾝ6下段(中間)切出し部ﾜｰｸ無
3546  LD      X6E  ; ﾚｰﾝ7上段(中間)切出し部ﾜｰｸ検出
      OUT     T194 K10  ; ﾚｰﾝ7上段(中間)切出し部ﾜｰｸ検出
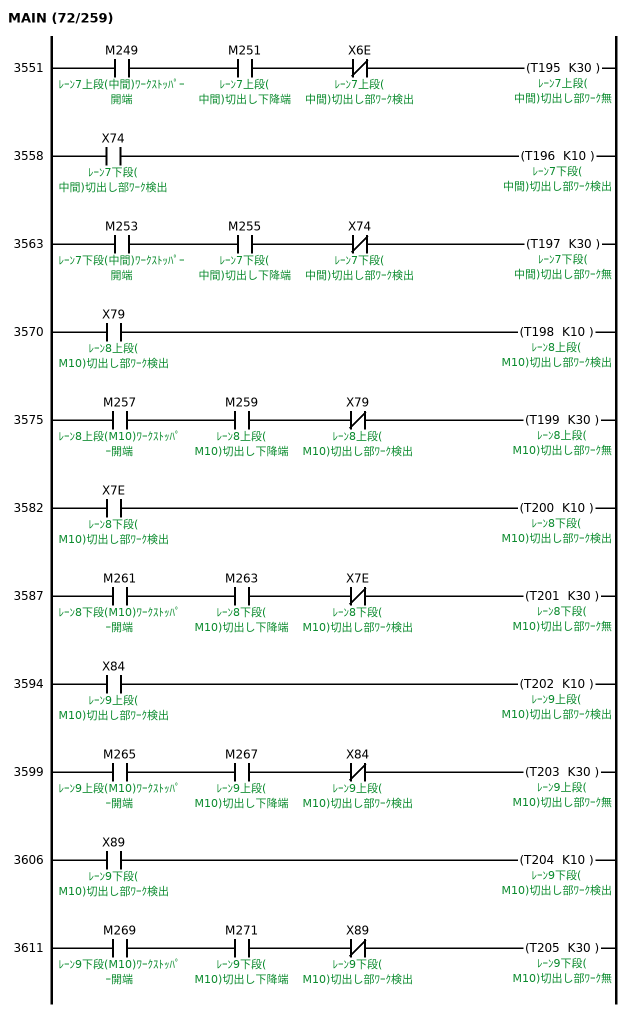
3551  LD      M249  ; ﾚｰﾝ7上段(中間)ﾜｰｸｽﾄｯﾊﾟｰ開端
      AND     M251  ; ﾚｰﾝ7上段(中間)切出し下降端
      ANI     X6E  ; ﾚｰﾝ7上段(中間)切出し部ﾜｰｸ検出
      OUT     T195 K30  ; ﾚｰﾝ7上段(中間)切出し部ﾜｰｸ無
3558  LD      X74  ; ﾚｰﾝ7下段(中間)切出し部ﾜｰｸ検出
      OUT     T196 K10  ; ﾚｰﾝ7下段(中間)切出し部ﾜｰｸ検出
3563  LD      M253  ; ﾚｰﾝ7下段(中間)ﾜｰｸｽﾄｯﾊﾟｰ開端
      AND     M255  ; ﾚｰﾝ7下段(中間)切出し下降端
      ANI     X74  ; ﾚｰﾝ7下段(中間)切出し部ﾜｰｸ検出
      OUT     T197 K30  ; ﾚｰﾝ7下段(中間)切出し部ﾜｰｸ無
3570  LD      X79  ; ﾚｰﾝ8上段(M10)切出し部ﾜｰｸ検出
      OUT     T198 K10  ; ﾚｰﾝ8上段(M10)切出し部ﾜｰｸ検出
3575  LD      M257  ; ﾚｰﾝ8上段(M10)ﾜｰｸｽﾄｯﾊﾟｰ開端
      AND     M259  ; ﾚｰﾝ8上段(M10)切出し下降端
      ANI     X79  ; ﾚｰﾝ8上段(M10)切出し部ﾜｰｸ検出
      OUT     T199 K30  ; ﾚｰﾝ8上段(M10)切出し部ﾜｰｸ無
3582  LD      X7E  ; ﾚｰﾝ8下段(M10)切出し部ﾜｰｸ検出
      OUT     T200 K10  ; ﾚｰﾝ8下段(M10)切出し部ﾜｰｸ検出
3587  LD      M261  ; ﾚｰﾝ8下段(M10)ﾜｰｸｽﾄｯﾊﾟｰ開端
      AND     M263  ; ﾚｰﾝ8下段(M10)切出し下降端
      ANI     X7E  ; ﾚｰﾝ8下段(M10)切出し部ﾜｰｸ検出
      OUT     T201 K30  ; ﾚｰﾝ8下段(M10)切出し部ﾜｰｸ無
3594  LD      X84  ; ﾚｰﾝ9上段(M10)切出し部ﾜｰｸ検出
      OUT     T202 K10  ; ﾚｰﾝ9上段(M10)切出し部ﾜｰｸ検出
3599  LD      M265  ; ﾚｰﾝ9上段(M10)ﾜｰｸｽﾄｯﾊﾟｰ開端
      AND     M267  ; ﾚｰﾝ9上段(M10)切出し下降端
      ANI     X84  ; ﾚｰﾝ9上段(M10)切出し部ﾜｰｸ検出
      OUT     T203 K30  ; ﾚｰﾝ9上段(M10)切出し部ﾜｰｸ無
3606  LD      X89  ; ﾚｰﾝ9下段(M10)切出し部ﾜｰｸ検出
      OUT     T204 K10  ; ﾚｰﾝ9下段(M10)切出し部ﾜｰｸ検出
3611  LD      M269  ; ﾚｰﾝ9下段(M10)ﾜｰｸｽﾄｯﾊﾟｰ開端
      AND     M271  ; ﾚｰﾝ9下段(M10)切出し下降端
      ANI     X89  ; ﾚｰﾝ9下段(M10)切出し部ﾜｰｸ検出
      OUT     T205 K30  ; ﾚｰﾝ9下段(M10)切出し部ﾜｰｸ無
